//  ================================================================================
//  OPTIONAL EDGE VALIDATIONS (if instrumentation available)
//  ================================================================================
//TEST_SingleTimeoutEvent_EmitsSingleTerminalTransition_NoDoubleFire();
//TEST_LastCommandCompletionTimeStamped_OnTimeoutComplete();
//TEST_ElapsedTimeReported_MatchesApproxTimeoutDuration();

METHOD PRIVATE TEST_Busy_FalseToTrue_OnStart_TrueToFalse_OnComplete
VAR_INST
	DynamicCycles : INT := 0;
END_VAR
VAR
	// Non FB or Interface instance variables
	TestName : Tc2_System.T_MaxString := 'TEST_Busy_FalseToTrue_OnStart_TrueToFalse_OnComplete';
	TestIdx : DINT := INDEX_TEST_BUSY_FALSETOTRUE_ONSTART_TRUETOFALSE_ONCOMPLETE;
	BusyWasTrue : BOOL := FALSE; // Track if we saw Busy=TRUE
END_VAR
TEST(__POUNAME());

// Purpose: Validates Busy flag transitions FALSE→TRUE on start, TRUE→FALSE on complete
// Based on logs: Busy changes at command start (cycle 1,618,132) and timeout complete (cycle 1,618,633)

// Initialize test objects on first cycle only
IF DynamicCycles = 0 THEN
	TestCommand[TestIdx].Initialize();
	TestComponent[TestIdx].Initialize();
	TestCommandConfig[TestIdx].Initialize();
	TestPermIntlk[TestIdx].Initialize();

	// Safe interface assignments
	iTestCommand := TestCommand[TestIdx];
	iTestCommandConfig := TestCommandConfig[TestIdx];
	iTestComponent := TestComponent[TestIdx];
	iTestPermIntlkConfig := TestPermIntlk[TestIdx];

	// Interface validation with protection
	IF iTestCommand = 0 THEN
		AssertTrue(Condition := FALSE, Message := 'TEST FAILED: iTestCommand interface is null');
		DynamicCycles := 0;
		RETURN;
	END_IF

	IF iTestCommandConfig = 0 THEN
		AssertTrue(Condition := FALSE, Message := 'TEST FAILED: iTestCommandConfig interface is null');
		DynamicCycles := 0;
		RETURN;
	END_IF

	IF iTestComponent = 0 THEN
		AssertTrue(Condition := FALSE, Message := 'TEST FAILED: iTestComponent interface is null');
		DynamicCycles := 0;
		RETURN;
	END_IF

	// Configure command to trigger timeout (no completion condition)
	iTestCommandConfig.P_CommandConfiguration.CommandDescription := 'Busy Flag Transition Test';
	iTestCommandConfig.P_CommandConfiguration.TimeoutTime := T#100MS; // Short timeout
	IF __ISVALIDREF(iTestCommandConfig.P_CommandConfiguration.BaseConfiguration) THEN
		iTestCommandConfig.P_CommandConfiguration.BaseConfiguration.LogTraceConfiguration.When := E_LogTraceWhen.xRunOnInitOnly;
	END_IF

	// Setup component to be enabled and not busy
	IF iTestComponent <> 0 THEN
		iTestComponent.P_ComponentStatus.BaseStatus.Enabled := TRUE;
		iTestComponent.P_ComponentStatus.BaseStatus.Busy := FALSE;
		iTestComponent.P_ComponentStatus.BaseStatus.Error := FALSE;
	END_IF

	// Configure permissive to be OK
	IF iTestPermIntlkConfig <> 0 THEN
		iTestPermIntlkConfig.P_PermIntlkConfiguration.PermIntlkObj[1].Description := 'Busy Transition Permissive';
		iTestPermIntlkConfig.P_PermIntlkConfiguration.PermIntlkObj[1].Condition := TRUE;
		iTestPermIntlkConfig.P_PermIntlkConfiguration.PermIntlkObj[1].Index := 1;
		TestPermIntlk[TestIdx].CyclicLogic(); // Update permissive evaluation
	END_IF

	// Setup command with configurations
	iTestCommand.InjectConfigurations(
		iComponent := iTestComponent,
		iCommandConfiguration := iTestCommandConfig,
		iPermIntlkConfiguration := iTestPermIntlkConfig
	);

	// Resolve configurations after injection
	iTestCommand.CyclicLogic();

	// Verify initial Busy is FALSE
	AssertFalse(
		Condition := iTestCommand.P_CommandStatus.BaseStatus.Busy,
		Message := 'Busy should be FALSE before Execute'
	);

	// Execute command
	iTestCommand.Execute();

	// Verify Execute() accepted the command
	AssertEquals_UDINT(
		Expected := E_CommandResult.Accepted,
		Actual := iTestCommand.P_CommandStatus.Result,
		Message := 'Execute() should set Result to Accepted'
	);
ELSE
	// Refresh interface references for subsequent cycles
	iTestCommand := TestCommand[TestIdx];
	iTestCommandConfig := TestCommandConfig[TestIdx];
END_IF

DynamicCycles := DynamicCycles + 1;

// Run cyclic logic
iTestCommand.CyclicLogic();

// Check Busy flag transitions
IF DynamicCycles = 1 THEN
	// After first cycle, Busy should be TRUE (FALSE→TRUE transition)
	AssertTrue(
		Condition := iTestCommand.P_CommandStatus.BaseStatus.Busy,
		Message := 'Busy should transition FALSE→TRUE on command start (cycle 1)'
	);
	BusyWasTrue := TRUE;
END_IF

// Track when Busy goes back to FALSE
IF BusyWasTrue AND NOT iTestCommand.P_CommandStatus.BaseStatus.Busy THEN
	// Busy transitioned TRUE→FALSE (timeout complete)
	AssertEquals_UDINT(
		Expected := E_CommandState.Complete,
		Actual := iTestCommand.P_CommandStatus.StepState,
		Message := 'When Busy transitions TRUE→FALSE, command should be in Complete state'
	);

	// Test passed, finish
	TEST_FINISHED();
END_IF

// Safety: Don't run forever if something goes wrong
IF DynamicCycles > 1000 THEN
	AssertTrue(Condition := FALSE, Message := 'TEST TIMEOUT: Command did not complete after 1000 cycles');
	TEST_FINISHED();
END_IF
END_METHOD

END_FUNCTION_BLOCK

// Tests/FB_LogTests
FUNCTION_BLOCK FB_LogTests EXTENDS TcUnit.FB_TestSuite
VAR
	// Array of test event log handlers - one for each test method
	TestEventLogHandlers : ARRAY[GC_Test.Index_TestFB_Logging_MIN..GC_Test.Index_TestFB_Logging_MAX] OF FB_EventLogHandler;

	// Test instance indices (for clarity and maintainability)
	IDX_FirstCycle					: DINT := 0;
	IDX_NormalOperation				: DINT := 1;
	IDX_BufferHasEntries			: DINT := 2;
	IDX_HighLoad					: DINT := 3;
	IDX_BufferNearCapacity			: DINT := 4;
	IDX_EmergencyFill				: DINT := 5;
	IDX_SuccessfulPersistence		: DINT := 6;
	IDX_FailureOnPersistence		: DINT := 7;
	IDX_RepeatedPersistenceFailures	: DINT := 8;
	IDX_MaxBackoffReached			: DINT := 9;
	IDX_NormalLoadBufferHealth		: DINT := 10;
	IDX_BufferOverflow				: DINT := 11;
	IDX_LogProcessing				: DINT := 12;
	IDX_MultipleCycles				: DINT := 13;
	IDX_ProcessingSeverity			: DINT := 14;
	IDX_TaskCycleExceed			: DINT := 15;
	IDX_TaskWithinLimits			: DINT := 16;
	IDX_AllTasksMonitored			: DINT := 17;
	IDX_EmptyBuffer					: DINT := 18;
	IDX_QueueOverflow				: DINT := 19;

	// Critical test indices
	IDX_PersistenceException		: DINT := 20;
	IDX_PersistenceBlocked			: DINT := 21;
	IDX_BufferNearFullCritical		: DINT := 22;
	IDX_BufferFullCritical			: DINT := 23;
	IDX_MaxDequeueLoad				: DINT := 24;
	IDX_HighJitter					: DINT := 25;
	IDX_ExtendedPersistenceFailure	: DINT := 26;
	IDX_Restart						: DINT := 27;
	IDX_ProcessingAllSeverities	: DINT := 28;
	IDX_OverflowCondition			: DINT := 29;

	// Robustness test indices
	IDX_BufferAtMaxCapacity		: DINT := 30;
	IDX_SustainedHighThroughput	: DINT := 31;
	IDX_MixedSeverityFlood			: DINT := 32;
	IDX_MaxDequeueRate				: DINT := 33;
	IDX_BackoffTimerActive			: DINT := 34;
	IDX_HeavyOSLoad					: DINT := 35;
	IDX_RepeatedPersistenceFailureRobust	: DINT := 36;
	IDX_PersistenceUnhandledException	: DINT := 37;
	IDX_BufferOverflowRecovered		: DINT := 38;
	IDX_MultipleTasksMonitored		: DINT := 39;

	// Note: We have exactly 40 slots (0-39) based on GC_Test configuration
END_VAR

// Core Functional Tests
GivenFirstCycle_WhenProgramRuns_ExpectInitializationComplete();
GivenNormalOperation_WhenLogDequeueCalled_ExpectEntriesProcessed();
GivenBufferHasEntries_WhenDequeueRuns_ExpectEntriesForwarded();
GivenHighLoad_WhenDequeueRuns_ExpectRateReduced();
GivenBufferNearCapacity_WhenDequeueRuns_ExpectRateIncreased();
GivenEmergencyFill_WhenDequeueRuns_ExpectMaxRateCappedAt200();
GivenSuccessfulPersistence_WhenAddToEventLog_ExpectTrueReturned();
GivenFailureOnPersistence_WhenAddToEventLog_ExpectFalseReturned();
GivenRepeatedPersistenceFailures_WhenHandleFailureCalled_ExpectExponentialBackoffApplied();
GivenMaxBackoffReached_WhenHandleFailureCalled_ExpectNoFurtherIncrease();
GivenNormalLoad_WhenUpdateBufferHealthMetrics_ExpectAccurateUtilization();
GivenBufferOverflow_WhenUpdateBufferHealthMetrics_ExpectOverflowCountIncremented();
GivenLogProcessing_WhenUpdatePerformanceMetrics_ExpectThroughputCalculated();
GivenMultipleCycles_WhenUpdatePerformanceMetrics_ExpectRollingAverageUpdated();
GivenProcessing_WhenUpdateSeverityMetrics_ExpectSeverityCountersCorrect();
GivenTaskCycleExceed_WhenMonitorPlcSystemRuns_ExpectCriticalEventLogged();
GivenTaskWithinLimits_WhenMonitorPlcSystemRuns_ExpectNoViolationLogged();
GivenAllTasksMonitored_WhenMonitorPlcSystemRuns_ExpectUtilizationPercentagesCalculated();
GivenEmptyBuffer_WhenLogDequeueCalled_ExpectNoErrors();
GivenQueueOverflow_WhenEnqueueCalled_ExpectOldestEntriesDroppedGracefully();

// High-Criticality Tests
GivenPersistenceThrowsException_WhenAddToEventLog_ExpectSafeRecovery();
GivenPersistenceBlocked_WhenHandleFailureRuns_ExpectProcessingSuspendedUntilTimeout();
GivenBufferNearFull_WhenCriticalAndDebugEntriesEnqueued_ExpectCriticalEntriesPreserved();
GivenBufferFull_WhenNewCriticalEntryArrives_ExpectSpaceReservedForCritical();
GivenMaxDequeueLoad_WhenCycleRuns_ExpectTaskNotToExceed50ms();
GivenHighJitter_WhenMonitoringTaskUtilization_ExpectCorrectHealthScoreLogged();
GivenExtendedPersistenceFailure_WhenRecovered_ExpectRateGraduallyRestored();
GivenRestart_WhenLoggerResumes_ExpectMetricsResetAndSafeStartup();
GivenProcessingAcrossAllSeverities_WhenMetricsUpdated_ExpectAccurateSeverityDistribution();
GivenOverflowCondition_WhenMetricsUpdated_ExpectDroppedCountAccurate();

// Stress and Robustness Tests
GivenBufferAtMaxCapacity_WhenFloodedWithEntries_ExpectGracefulDegradation();
GivenSustainedHighThroughput_WhenRunningFor10Minutes_ExpectNoMemoryLeakOrCycleExceed();
GivenMixedSeverityFlood_WhenProcessing_ExpectLatencyForCriticalEntriesLow();
GivenMaxDequeueRate_WhenCycleRuns_ExpectCycleTimeWithin50msBudget();
GivenBackoffTimerActive_WhenNextCycleRuns_ExpectNoPrematureRetries();
GivenHeavyOSLoad_WhenPersistenceSlows_ExpectLoggerTaskStillMeetsCycleTime();
GivenRepeatedPersistenceFailure_WhenRecovered_ExpectRateRestoredToNormal();
GivenPersistenceThrowsUnhandledException_WhenCaught_ExpectNoTaskCrash();
GivenBufferOverflow_WhenRecovered_ExpectMetricsReflectCorrectDropCounts();
GivenMultipleTasksMonitored_WhenSystemStable_ExpectUtilizationReportedAccurately();
GivenCycleExceeds_WhenDetected_ExpectHealthScoreReducedAndViolationLogged();
GivenSeverityMix_WhenProcessing_ExpectSeverityDistributionAccurate();

METHOD PRIVATE GivenAllTasksMonitored_WhenMonitorPlcSystemRuns_ExpectUtilizationPercentagesCalculated
VAR
END_VAR
TEST(__POUNAME());

//Assertions

TEST_FINISHED();
END_METHOD

METHOD PRIVATE GivenBufferHasEntries_WhenDequeueRuns_ExpectEntriesForwarded
VAR
	TestHandler				: REFERENCE TO FB_EventLogHandler;
	InitialBufferCount		: UDINT;
	FinalBufferCount		: UDINT;
	i						: INT;
	EntriesAdded			: INT := 10;
	ExpectedProcessed		: UDINT;
	ActualProcessed			: UDINT;
END_VAR
TEST(__POUNAME());

// Get reference to test instance for this test
TestHandler REF= TestEventLogHandlers[IDX_BufferHasEntries];

// Configure test instance for test mode
IF __ISVALIDREF(TestHandler.P_EventLogHandlerConfiguration.BaseConfiguration) THEN
	TestHandler.P_EventLogHandlerConfiguration.BaseConfiguration.InSimulation := TRUE;
ELSE
	TestHandler.Initialize();
END_IF

// Initialize the test handler and system components
TestHandler.Initialize();
GVL_System.RingBufferLog.Initialize();
GVL_System.GlobalEventLog.Initialize();

// Call CyclicLogic to process initialization
TestHandler.CyclicLogic();

// Ensure clean state
GVL_System.RingBufferLog.ClearBuffer();

// Arrange - Add entries to the buffer
InitialBufferCount := GVL_System.RingBufferLog.P_RingBufferStatus.ObjectCountInBufferPrim;

// Add test entries to buffer
FOR i := 1 TO EntriesAdded DO
	GVL_System.RingBufferLog.TraceWithSeverity(
		Message := CONCAT('Entry to forward #', INT_TO_STRING(i)),
		Severity := Global.TcEventSeverity.Info
	);
END_FOR

// Verify entries were added to buffer
AssertEquals_UDINT(
	Expected := InitialBufferCount + INT_TO_UDINT(EntriesAdded),
	Actual := GVL_System.RingBufferLog.P_RingBufferStatus.ObjectCountInBufferPrim,
	Message := 'Entries should be added to buffer before dequeue'
);

// Store the initial processed count
ActualProcessed := TestHandler.P_EventLogHandlerStatus.LoggingMetrics.TotalEntriesProcessed;

// Act - Run CyclicLogic which will dequeue and forward entries
TestHandler.CyclicLogic();

// Get final state
FinalBufferCount := GVL_System.RingBufferLog.P_RingBufferStatus.ObjectCountInBufferPrim;
ActualProcessed := TestHandler.P_EventLogHandlerStatus.LogCountThisScan;

// Assert - Verify entries were removed from buffer
AssertTrue(
	Condition := FinalBufferCount < InitialBufferCount + INT_TO_UDINT(EntriesAdded),
	Message := 'Buffer count should decrease after dequeue'
);

// Verify entries were actually processed (forwarded)
AssertTrue(
	Condition := ActualProcessed > 0,
	Message := 'Entries should be processed (forwarded) during dequeue'
);

// Calculate expected processed based on dynamic rate limits
ExpectedProcessed := MIN(INT_TO_UDINT(EntriesAdded),
                         UINT_TO_UDINT(TestHandler.P_EventLogHandlerStatus.DynamicMaxEntries));

// Verify we didn't exceed the dynamic rate limit
AssertTrue(
	Condition := ActualProcessed <= UINT_TO_UDINT(TestHandler.P_EventLogHandlerStatus.DynamicMaxEntries),
	Message := 'Should not process more than DynamicMaxEntries in one scan'
);

// Verify the number of entries removed matches the number processed
AssertEquals_UDINT(
	Expected := ActualProcessed,
	Actual := (InitialBufferCount + INT_TO_UDINT(EntriesAdded)) - FinalBufferCount,
	Message := 'Number of entries removed from buffer should match number processed'
);

// Verify metrics were updated
AssertEquals_UDINT(
	Expected := ActualProcessed,
	Actual := UINT_TO_UDINT(TestHandler.P_EventLogHandlerStatus.LoggingMetrics.EntriesProcessedThisCycle),
	Message := 'EntriesProcessedThisCycle should match actual processed count'
);

// Verify total entries processed was incremented
AssertTrue(
	Condition := TestHandler.P_EventLogHandlerStatus.LoggingMetrics.TotalEntriesProcessed >= ActualProcessed,
	Message := 'TotalEntriesProcessed should be incremented'
);

// Verify no errors during forwarding
AssertFalse(
	Condition := TestHandler.P_EventLogHandlerStatus.BaseStatus.Error,
	Message := 'No errors should occur during normal forwarding operation'
);

// Verify buffer health metrics were updated
AssertTrue(
	Condition := TestHandler.P_EventLogHandlerStatus.LoggingMetrics.BufferUtilizationPercentage >= 0.0,
	Message := 'Buffer utilization should be calculated after dequeue'
);

TEST_FINISHED();
END_METHOD

METHOD PRIVATE GivenBufferNearCapacity_WhenDequeueRuns_ExpectRateIncreased
VAR
	TestHandler				: REFERENCE TO FB_EventLogHandler;
	BufferCapacity			: UDINT;
	EntriesToAdd			: UDINT;
	NormalRate				: UINT;
	IncreasedRate			: UINT;
	i						: DINT;
	InitialBufferCount		: UDINT;
	FinalBufferCount		: UDINT;
	EntriesProcessed		: UDINT;
END_VAR
TEST(__POUNAME());

// Get reference to test instance for this test
TestHandler REF= TestEventLogHandlers[IDX_BufferNearCapacity];

// Configure test instance - enable metrics tracking

// Initialize the test handler and system components
TestHandler.Initialize();
GVL_System.RingBufferLog.Initialize();
GVL_System.GlobalEventLog.Initialize();

// Call CyclicLogic to process initialization
TestHandler.CyclicLogic();

// Ensure clean state
GVL_System.RingBufferLog.ClearBuffer();

// Get buffer capacity
BufferCapacity := GVL_System.RingBufferLog.P_RingBufferStatus.BufferCapacity;

// Arrange - Set low task utilization (so rate increase is based on buffer, not task load)
GVL_System.PlcSystemInfo[GPL_BASE.INDEX_LOG_TASK].TaskUtilizationPercentage := 0.2; // 20% utilization

// Calculate normal rate with empty buffer
NormalRate := TestHandler.CalculateDynamicRate();

// Verify we're at normal rate with low load and empty buffer
AssertEquals_UINT(
	Expected := UDINT_TO_UINT(GPL_Base.MAX_LOG_ENTRIES_PER_SCAN),
	Actual := NormalRate,
	Message := 'Low load with empty buffer should use normal rate'
);

// Fill buffer to near capacity (80% full - should trigger rate increase)
EntriesToAdd := (BufferCapacity * 80) / 100;  // 80% of capacity

FOR i := 1 TO UDINT_TO_DINT(EntriesToAdd) DO
	GVL_System.RingBufferLog.TraceWithSeverity(
		Message := CONCAT('Buffer fill test entry ', DINT_TO_STRING(i)),
		Severity := Global.TcEventSeverity.Info
	);
END_FOR

InitialBufferCount := GVL_System.RingBufferLog.P_RingBufferStatus.ObjectCountInBufferPrim;

// Verify buffer is near capacity
AssertTrue(
	Condition := InitialBufferCount >= (BufferCapacity * 75) / 100,
	Message := 'Buffer should be at least 75% full for this test'
);

// Act - Calculate rate with near-full buffer
IncreasedRate := TestHandler.CalculateDynamicRate();

// Assert - Rate should be increased when buffer is near capacity
AssertTrue(
	Condition := IncreasedRate > NormalRate,
	Message := 'Processing rate should increase when buffer is near capacity'
);

// Specifically, when buffer > 75% and low task load, rate should double
AssertEquals_UINT(
	Expected := UDINT_TO_UINT(GPL_Base.MAX_LOG_ENTRIES_PER_SCAN * 2),
	Actual := IncreasedRate,
	Message := 'Buffer near capacity with low load should double the rate'
);

// Verify the increased rate doesn't exceed emergency maximum
AssertTrue(
	Condition := IncreasedRate <= UDINT_TO_UINT(200),
	Message := 'Increased rate should not exceed emergency maximum'
);

// Call CyclicLogic to process with increased rate
TestHandler.CyclicLogic();

// Get final state
FinalBufferCount := GVL_System.RingBufferLog.P_RingBufferStatus.ObjectCountInBufferPrim;
EntriesProcessed := TestHandler.P_EventLogHandlerStatus.LogCountThisScan;

// Verify more entries were processed with increased rate
AssertTrue(
	Condition := EntriesProcessed > UINT_TO_UDINT(NormalRate),
	Message := 'Should process more entries when rate is increased'
);

// Verify buffer was reduced
AssertTrue(
	Condition := FinalBufferCount < InitialBufferCount,
	Message := 'Buffer count should decrease after processing with increased rate'
);

// Test emergency fill level (>90%)
GVL_System.RingBufferLog.ClearBuffer();
EntriesToAdd := (BufferCapacity * 95) / 100;  // 95% of capacity

FOR i := 1 TO UDINT_TO_DINT(EntriesToAdd) DO
	GVL_System.RingBufferLog.TraceWithSeverity(
		Message := CONCAT('Emergency fill test ', DINT_TO_STRING(i)),
		Severity := Global.TcEventSeverity.Critical
	);
END_FOR

// Calculate rate with emergency fill level
IncreasedRate := TestHandler.CalculateDynamicRate();

// Should be at emergency maximum
AssertEquals_UINT(
	Expected := UDINT_TO_UINT(200),
	Actual := IncreasedRate,
	Message := 'Emergency fill level should trigger maximum processing rate'
);

TEST_FINISHED();
END_METHOD

METHOD PRIVATE GivenBufferOverflow_WhenUpdateBufferHealthMetrics_ExpectOverflowCountIncremented
VAR
	InitialOverflowCount		: UDINT;
	FinalOverflowCount			: UDINT;
	BufferCapacity				: UDINT;
	i							: DINT;
	TestBufferFull				: BOOL;
END_VAR
TEST(__POUNAME());

// Initialize if needed
IF GVL_System.PlcSystemInfo[GPL_Base.INDEX_LOG_TASK].FirstCycle THEN
    GVL_System.RingBufferLog.Initialize();
    GVL_System.GlobalEventLog.Initialize();
    RETURN;
END_IF;

// Arrange - Get initial state
InitialOverflowCount := GVL_System.EventLogHandler.P_EventLogHandlerStatus.LoggingMetrics.BufferOverflowCount;
BufferCapacity := GVL_System.RingBufferLog.P_RingBufferStatus.BufferCapacity;

// Clear the buffer first
GVL_System.RingBufferLog.ClearBuffer();

// Fill the buffer to capacity
FOR i := 1 TO UDINT_TO_DINT(BufferCapacity) + 10 DO
	GVL_System.RingBufferLog.TraceWithSeverity(
		Message := CONCAT('Overflow test entry ', DINT_TO_STRING(i)),
		Severity := Global.TcEventSeverity.Info
	);
END_FOR;

// Verify buffer is full
TestBufferFull := GVL_System.RingBufferLog.P_RingBufferStatus.BufferIsFullPrim;
AssertTrue(
	Condition := TestBufferFull,
	Message := 'Buffer should be full after adding more entries than capacity'
);

// Act - Call UpdateBufferHealthMetrics multiple times while buffer is full
GVL_System.EventLogHandler.UpdateBufferHealthMetrics();  // First call - should increment
GVL_System.EventLogHandler.UpdateBufferHealthMetrics();  // Second call - should NOT increment (edge detection)
GVL_System.EventLogHandler.UpdateBufferHealthMetrics();  // Third call - should NOT increment

FinalOverflowCount := GVL_System.EventLogHandler.P_EventLogHandlerStatus.LoggingMetrics.BufferOverflowCount;

// Assert - Overflow count should increment only once due to edge detection
AssertEquals_UDINT(
	Expected := InitialOverflowCount + 1,
	Actual := FinalOverflowCount,
	Message := 'Overflow count should increment only once on rising edge of buffer full'
);

// Clear some entries to make buffer not full
// Call LogDequeue multiple times to ensure buffer is drained enough
FOR i := 1 TO 10 DO
	GVL_System.EventLogHandler.LogDequeue();
	IF NOT GVL_System.RingBufferLog.P_RingBufferStatus.BufferIsFullPrim THEN
		EXIT; // Buffer is no longer full, stop dequeuing
	END_IF;
END_FOR;

// Reset the edge trigger by having buffer not full
TestBufferFull := GVL_System.RingBufferLog.P_RingBufferStatus.BufferIsFullPrim;
AssertFalse(
	Condition := TestBufferFull,
	Message := 'Buffer should not be full after dequeue'
);

// Fill again to test another edge
FOR i := 1 TO 100 DO
	GVL_System.RingBufferLog.TraceWithSeverity(
		Message := CONCAT('Second overflow test ', DINT_TO_STRING(i)),
		Severity := Global.TcEventSeverity.Critical
	);
END_FOR;

// Call UpdateBufferHealthMetrics again with new overflow
GVL_System.EventLogHandler.UpdateBufferHealthMetrics();

// Should increment again on new rising edge
AssertEquals_UDINT(
	Expected := InitialOverflowCount + 2,
	Actual := GVL_System.EventLogHandler.P_EventLogHandlerStatus.LoggingMetrics.BufferOverflowCount,
	Message := 'Overflow count should increment on each new rising edge'
);

TEST_FINISHED();
END_METHOD

METHOD PRIVATE GivenEmergencyFill_WhenDequeueRuns_ExpectMaxRateCappedAt200
VAR
END_VAR
TEST(__POUNAME());

//Assertions

TEST_FINISHED();
END_METHOD

METHOD PRIVATE GivenEmptyBuffer_WhenLogDequeueCalled_ExpectNoErrors
VAR
	TestHandler					: REFERENCE TO FB_EventLogHandler;
	InitialErrorState			: BOOL;
	FinalErrorState				: BOOL;
	InitialProcessedCount		: UDINT;
	FinalProcessedCount			: UDINT;
	BufferCountBeforeDequeue	: UDINT;
	BufferCountAfterDequeue	: UDINT;
END_VAR
TEST(__POUNAME());

// Get reference to test instance for this test
TestHandler REF= TestEventLogHandlers[IDX_EmptyBuffer];

// Configure test instance - enable metrics tracking

// Initialize the test handler and system components
TestHandler.Initialize();
GVL_System.RingBufferLog.Initialize();
GVL_System.GlobalEventLog.Initialize();

// Call CyclicLogic to process initialization
TestHandler.CyclicLogic();

// Ensure buffer is completely empty
GVL_System.RingBufferLog.ClearBuffer();

// Verify buffer is empty
AssertEquals_UDINT(
	Expected := 0,
	Actual := GVL_System.RingBufferLog.P_RingBufferStatus.ObjectCountInBufferPrim,
	Message := 'Buffer should be empty before test'
);

// Get initial state
InitialErrorState := TestHandler.P_EventLogHandlerStatus.BaseStatus.Error;
InitialProcessedCount := TestHandler.P_EventLogHandlerStatus.LoggingMetrics.TotalEntriesProcessed;
BufferCountBeforeDequeue := GVL_System.RingBufferLog.P_RingBufferStatus.ObjectCountInBufferPrim;

// Verify no errors initially
AssertFalse(
	Condition := InitialErrorState,
	Message := 'Should start with no errors'
);

// Act - Call LogDequeue on empty buffer (should handle gracefully)
TestHandler.LogDequeue();

// Get final state
FinalErrorState := TestHandler.P_EventLogHandlerStatus.BaseStatus.Error;
FinalProcessedCount := TestHandler.P_EventLogHandlerStatus.LoggingMetrics.TotalEntriesProcessed;
BufferCountAfterDequeue := GVL_System.RingBufferLog.P_RingBufferStatus.ObjectCountInBufferPrim;

// Assert - No errors should occur
AssertFalse(
	Condition := FinalErrorState,
	Message := 'No errors should occur when dequeuing from empty buffer'
);

// Buffer should remain empty
AssertEquals_UDINT(
	Expected := 0,
	Actual := BufferCountAfterDequeue,
	Message := 'Buffer should remain empty'
);

// No entries should be processed
AssertEquals_UDINT(
	Expected := InitialProcessedCount,
	Actual := FinalProcessedCount,
	Message := 'No entries should be processed from empty buffer'
);

// LogCountThisScan should be 0
AssertEquals_UDINT(
	Expected := 0,
	Actual := TestHandler.P_EventLogHandlerStatus.LogCountThisScan,
	Message := 'LogCountThisScan should be 0 for empty buffer'
);

// Test multiple dequeue calls on empty buffer (should all handle gracefully)
TestHandler.LogDequeue();
TestHandler.LogDequeue();
TestHandler.LogDequeue();

// Still no errors
AssertFalse(
	Condition := TestHandler.P_EventLogHandlerStatus.BaseStatus.Error,
	Message := 'Multiple dequeue calls on empty buffer should not cause errors'
);

// Call full CyclicLogic on empty buffer (should handle gracefully)
TestHandler.CyclicLogic();

// Verify no errors after full cycle
AssertFalse(
	Condition := TestHandler.P_EventLogHandlerStatus.BaseStatus.Error,
	Message := 'Full CyclicLogic on empty buffer should not cause errors'
);

// Verify metrics remain stable
AssertEquals_UDINT(
	Expected := 0,
	Actual := TestHandler.P_EventLogHandlerStatus.LoggingMetrics.EntriesProcessedThisCycle,
	Message := 'EntriesProcessedThisCycle should be 0 for empty buffer'
);

// Buffer utilization should be 0%
AssertEquals_REAL(
	Expected := 0.0,
	Actual := TestHandler.P_EventLogHandlerStatus.LoggingMetrics.BufferUtilizationPercentage,
	Delta := 0.01,
	Message := 'Buffer utilization should be 0% when empty'
);

// Dynamic rate calculation should still work
AssertTrue(
	Condition := TestHandler.CalculateDynamicRate() > 0,
	Message := 'Dynamic rate calculation should work even with empty buffer'
);

// No persistence failures should occur
AssertEquals_UINT(
	Expected := 0,
	Actual := TestHandler.P_EventLogHandlerStatus.BackoffState.PersistenceFailureCount,
	Message := 'No persistence failures should occur with empty buffer'
);

// System health should be good
AssertTrue(
	Condition := TestHandler.P_EventLogHandlerStatus.LoggingMetrics.SystemHealthScore >= 90.0,
	Message := 'System health should be high with empty buffer and no errors'
);

TEST_FINISHED();
END_METHOD

METHOD PRIVATE GivenFailureOnPersistence_WhenAddToEventLog_ExpectFalseReturned
VAR
	TestHandler				: REFERENCE TO FB_EventLogHandler;
	PersistenceResult		: BOOL;
	InitialSuccessCount		: UDINT;
	FinalSuccessCount		: UDINT;
	InitialFailureCount		: UINT;
	FinalFailureCount		: UINT;
END_VAR
TEST(__POUNAME());

// Get reference to test instance for this test
TestHandler REF= TestEventLogHandlers[IDX_FailureOnPersistence];

// Configure test instance for TEST MODE to simulate failure
IF __ISVALIDREF(TestHandler.P_EventLogHandlerConfiguration.BaseConfiguration) THEN
	TestHandler.P_EventLogHandlerConfiguration.BaseConfiguration.InSimulation := TRUE;
ELSE
	TestHandler.Initialize();
END_IF

// Initialize the test handler and system components
TestHandler.Initialize();
GVL_System.RingBufferLog.Initialize();
GVL_System.GlobalEventLog.Initialize();

// Call CyclicLogic to process initialization
TestHandler.CyclicLogic();

// Ensure clean state
GVL_System.RingBufferLog.ClearBuffer();

// Get initial metrics
InitialFailureCount := TestHandler.P_EventLogHandlerStatus.BackoffState.PersistenceFailureCount;

// Arrange - Simulate a persistence failure condition
// Since we're in test mode, we need to mock the failure
// This would require setting up the test status to simulate failure
TestHandler.P_EventLogHandlerStatus.BackoffState.PersistenceBlocked := TRUE;

// Add a test entry to the buffer
GVL_System.RingBufferLog.TraceWithSeverity(
	Message := 'Test entry for failed persistence',
	Severity := Global.TcEventSeverity.Error
);

// Verify entry was added
AssertEquals_UDINT(
	Expected := 1,
	Actual := GVL_System.RingBufferLog.P_RingBufferStatus.ObjectCountInBufferPrim,
	Message := 'One entry should be in buffer'
);

// Act - Try to add to event log when persistence is blocked
// First, remove from buffer to make available in P_LastObjectRemoved
GVL_System.RingBufferLog.RemoveObject();

// Now try to add it to the event log (should fail due to PersistenceBlocked)
PersistenceResult := TestHandler.AddToEventLog();

// Assert - Verify failed persistence
AssertFalse(
	Condition := PersistenceResult,
	Message := 'AddToEventLog should return FALSE when persistence is blocked'
);

// Get final metrics
FinalFailureCount := TestHandler.P_EventLogHandlerStatus.BackoffState.PersistenceFailureCount;

// Success count verification removed as PersistenceSuccessCount metric doesn't exist

// Reset persistence blocked to test normal failure handling
TestHandler.P_EventLogHandlerStatus.BackoffState.PersistenceBlocked := FALSE;

// Simulate a different type of failure - we could mock the GlobalEventLog to fail
// For this test, we'll simulate by checking the behavior when AddToEventLog
// is called but the operation fails (returns FALSE)

// Add another entry
GVL_System.RingBufferLog.TraceWithSeverity(
	Message := 'Test entry for simulated add failure',
	Severity := Global.TcEventSeverity.Critical
);

// Process it
GVL_System.RingBufferLog.RemoveObject();

// In test mode, we can force AddToEventLog to return FALSE
// by manipulating the test status - this simulates GlobalEventLog failure
// Note: This assumes AddToEventLog checks some condition we can control
// If not, we'd need a method to simulate GlobalEventLog failures

// Call HandlePersistenceFailure to simulate what happens on failure
TestHandler.HandlePersistenceFailure();

// Verify failure handling was activated
AssertTrue(
	Condition := TestHandler.P_EventLogHandlerStatus.BackoffState.PersistenceBlocked,
	Message := 'Persistence should be blocked after handling failure'
);

// Verify backoff delay was set
AssertTrue(
	Condition := TestHandler.P_EventLogHandlerStatus.BackoffState.BackoffDelayMs >= 100,
	Message := 'Backoff delay should be set after failure'
);

// Verify failure count incremented
AssertTrue(
	Condition := TestHandler.P_EventLogHandlerStatus.BackoffState.PersistenceFailureCount > 0,
	Message := 'PersistenceFailureCount should increment after failure'
);

// Backoff timer check removed as BackoffStartTime property doesn't exist

TEST_FINISHED();
END_METHOD

METHOD PRIVATE GivenFirstCycle_WhenProgramRuns_ExpectInitializationComplete
VAR
	// Local test variables
	PreInitBufferCount		: UDINT;
	PostInitBufferCount		: UDINT;
	TestHandler				: REFERENCE TO FB_EventLogHandler;
END_VAR
TEST(__POUNAME());

// Get reference to test instance for this test
TestHandler REF= TestEventLogHandlers[IDX_FirstCycle];

// Configure test instance for test mode
IF __ISVALIDREF(TestHandler.P_EventLogHandlerConfiguration.BaseConfiguration) THEN
	TestHandler.P_EventLogHandlerConfiguration.BaseConfiguration.InSimulation := TRUE;
ELSE
	TestHandler.Initialize();
END_IF

// Configure test instance settings

// Initialize the test instance
TestHandler.Initialize();

// Call CyclicLogic to process initialization
TestHandler.CyclicLogic();

// Arrange - Clear any existing state and store pre-init values
GVL_System.RingBufferLog.ClearBuffer();
PreInitBufferCount := GVL_System.RingBufferLog.P_RingBufferStatus.ObjectCountInBufferPrim;

// Act - Simulate what the EventLogHandler does on first cycle:
// Initialize both the RingBufferLog and GlobalEventLog
GVL_System.RingBufferLog.Initialize();
GVL_System.GlobalEventLog.Initialize();
PostInitBufferCount := GVL_System.RingBufferLog.P_RingBufferStatus.ObjectCountInBufferPrim;

// Verify the test handler is initialized
AssertTrue(
	Condition := TestHandler.P_EventLogHandlerStatus.BaseStatus.Initialized,
	Message := 'Test EventLogHandler should be initialized'
);

// Assert - Verify components are properly initialized
AssertTrue(
	Condition := __ISVALIDREF(GVL_System.RingBufferLog.P_RingBufferStatus.BaseStatus) AND
	             GVL_System.RingBufferLog.P_RingBufferStatus.BaseStatus.Initialized,
	Message := 'RingBufferLog should be initialized after first cycle behavior'
);

AssertTrue(
	Condition := GVL_System.GlobalEventLog.P_BaseStatus.Initialized,
	Message := 'GlobalEventLog should be initialized after first cycle behavior'
);

// Verify ring buffer is ready for dequeue operations
AssertEquals_UDINT(
	Expected := 0,
	Actual := PostInitBufferCount,
	Message := 'RingBufferLog should be empty and ready for entries after initialization'
);

// Verify buffer has proper capacity configured
AssertTrue(
	Condition := GVL_System.RingBufferLog.P_RingBufferStatus.BufferCapacity > 0,
	Message := 'RingBufferLog must have a positive capacity to accept log entries'
);

// Verify no error states that would prevent dequeue operations
AssertFalse(
	Condition := __ISVALIDREF(GVL_System.RingBufferLog.P_RingBufferStatus.BaseStatus) AND
	             GVL_System.RingBufferLog.P_RingBufferStatus.BaseStatus.Error,
	Message := 'No errors should be present that would block dequeue operations'
);

AssertFalse(
	Condition := GVL_System.RingBufferLog.P_RingBufferStatus.BufferIsFullPrim,
	Message := 'Buffer should not report full state after initialization'
);

// Verify global event log has no errors that would prevent receiving entries
AssertFalse(
	Condition := GVL_System.GlobalEventLog.P_BaseStatus.Error,
	Message := 'GlobalEventLog should have no errors that would prevent receiving dequeued entries'
);

// Verify test handler configuration is in test mode
IF __ISVALIDREF(TestHandler.P_EventLogHandlerConfiguration.BaseConfiguration) THEN
	AssertTrue(
		Condition := TestHandler.P_EventLogHandlerConfiguration.BaseConfiguration.InSimulation,
		Message := 'EventLogHandler should be in test mode'
	);
ELSE
	AssertTrue(
		Condition := FALSE,
		Message := 'EventLogHandlerConfiguration reference is invalid - cannot verify test mode'
	);
END_IF

// Verify test handler metrics are initialized
AssertEquals_UDINT(
	Expected := 0,
	Actual := TestHandler.P_EventLogHandlerStatus.LoggingMetrics.TotalEntriesProcessed,
	Message := 'Total entries processed should be 0 after initialization'
);

AssertEquals_REAL(
	Expected := 100.0,
	Actual := TestHandler.P_EventLogHandlerStatus.LoggingMetrics.SystemHealthScore,
	Delta := 0.01,
	Message := 'System health score should be 100% after initialization'
);

TEST_FINISHED();
END_METHOD

METHOD PRIVATE GivenHighLoad_WhenDequeueRuns_ExpectRateReduced
VAR
	TestHandler					: REFERENCE TO FB_EventLogHandler;
	SimulatedHighUtilization	: REAL := 0.85;  // 85% utilization
	SimulatedNormalUtilization	: REAL := 0.30;  // 30% utilization
	NormalMaxEntries			: UINT;
	HighLoadMaxEntries			: UINT;
	i							: INT;
	InitialBufferCount			: UDINT;
	FinalBufferCount			: UDINT;
	EntriesProcessed			: UDINT;
END_VAR
TEST(__POUNAME());

// Get reference to test instance for this test
TestHandler REF= TestEventLogHandlers[IDX_HighLoad];

// Configure test instance for test mode
IF __ISVALIDREF(TestHandler.P_EventLogHandlerConfiguration.BaseConfiguration) THEN
	TestHandler.P_EventLogHandlerConfiguration.BaseConfiguration.InSimulation := TRUE;
ELSE
	TestHandler.Initialize();
END_IF

// Initialize the test handler and system components
TestHandler.Initialize();
GVL_System.RingBufferLog.Initialize();
GVL_System.GlobalEventLog.Initialize();

// Call CyclicLogic to process initialization
TestHandler.CyclicLogic();

// Ensure clean state
GVL_System.RingBufferLog.ClearBuffer();

// Arrange - Set up normal load condition first
GVL_System.PlcSystemInfo[GPL_BASE.INDEX_LOG_TASK].TaskUtilizationPercentage := SimulatedNormalUtilization;

// Calculate normal rate by calling CalculateDynamicRate
NormalMaxEntries := TestHandler.CalculateDynamicRate();

// Verify normal rate is at expected level
AssertEquals_UINT(
	Expected := UDINT_TO_UINT(GPL_Base.MAX_LOG_ENTRIES_PER_SCAN),
	Actual := NormalMaxEntries,
	Message := 'Normal load should allow full processing rate'
);

// Now simulate high load condition
GVL_System.PlcSystemInfo[GPL_BASE.INDEX_LOG_TASK].TaskUtilizationPercentage := SimulatedHighUtilization;

// Add many entries to process
FOR i := 1 TO 50 DO
	GVL_System.RingBufferLog.TraceWithSeverity(
		Message := CONCAT('High load test entry ', INT_TO_STRING(i)),
		Severity := Global.TcEventSeverity.Warning
	);
END_FOR

InitialBufferCount := GVL_System.RingBufferLog.P_RingBufferStatus.ObjectCountInBufferPrim;

// Act - Calculate dynamic rate under high load
HighLoadMaxEntries := TestHandler.CalculateDynamicRate();

// Assert - Rate should be reduced under high load
AssertTrue(
	Condition := HighLoadMaxEntries < NormalMaxEntries,
	Message := 'Processing rate should be reduced under high load'
);

// When utilization > LOG_CYCLE_EXCEED_MAX_THRESHOLD (0.75), rate should be quartered
AssertEquals_UINT(
	Expected := UDINT_TO_UINT(GPL_Base.MAX_LOG_ENTRIES_PER_SCAN / 4),
	Actual := HighLoadMaxEntries,
	Message := 'High load (>75%) should reduce rate to quarter of normal'
);

// Store the calculated rate in the test handler's status
TestHandler.P_EventLogHandlerStatus.DynamicMaxEntries := HighLoadMaxEntries;

// Call CyclicLogic to process with the high load condition
TestHandler.CyclicLogic();

// Get final state
FinalBufferCount := GVL_System.RingBufferLog.P_RingBufferStatus.ObjectCountInBufferPrim;
EntriesProcessed := TestHandler.P_EventLogHandlerStatus.LogCountThisScan;

// Verify it respects the reduced rate limit
AssertTrue(
	Condition := EntriesProcessed <= UINT_TO_UDINT(HighLoadMaxEntries),
	Message := 'Should not process more than reduced rate limit under high load'
);

// Verify that entries were actually processed (but at reduced rate)
AssertTrue(
	Condition := EntriesProcessed > 0 AND EntriesProcessed <= UINT_TO_UDINT(HighLoadMaxEntries),
	Message := 'Should process some entries but respect high load limit'
);

// Verify buffer count decreased by the amount processed
AssertEquals_UDINT(
	Expected := InitialBufferCount - EntriesProcessed,
	Actual := FinalBufferCount,
	Message := 'Buffer should decrease by exactly the number of entries processed'
);

// Test moderate load (between 50% and 75%)
GVL_System.PlcSystemInfo[GPL_BASE.INDEX_LOG_TASK].TaskUtilizationPercentage := 0.6; // 60% utilization
NormalMaxEntries := TestHandler.CalculateDynamicRate();

// Should be half rate for moderate load
AssertEquals_UINT(
	Expected := UDINT_TO_UINT(GPL_Base.MAX_LOG_ENTRIES_PER_SCAN / 2),
	Actual := NormalMaxEntries,
	Message := 'Moderate load (50-75%) should reduce rate to half of normal'
);

TEST_FINISHED();
END_METHOD

METHOD PRIVATE GivenLogProcessing_WhenUpdatePerformanceMetrics_ExpectThroughputCalculated
VAR
END_VAR
TEST(__POUNAME());

//Assertions

TEST_FINISHED();
END_METHOD

METHOD PRIVATE GivenMaxBackoffReached_WhenHandleFailureCalled_ExpectNoFurtherIncrease
VAR
END_VAR
TEST(__POUNAME());

//Assertions

TEST_FINISHED();
END_METHOD

METHOD PRIVATE GivenMultipleCycles_WhenUpdatePerformanceMetrics_ExpectRollingAverageUpdated
VAR
	TestHandler					: REFERENCE TO FB_EventLogHandler;
	InitialAverage				: REAL;
	PreviousAverage				: REAL;
	CurrentAverage				: REAL;
	i							: INT;
	j							: INT;
	NumCycles					: INT := 10;
	EntriesPerCycle				: INT := 5;
	AverageChanged				: BOOL := FALSE;
	PeakTime					: UDINT;
END_VAR
TEST(__POUNAME());

// Get reference to test instance for this test
TestHandler REF= TestEventLogHandlers[IDX_MultipleCycles];

// Configure test instance - enable performance metrics

// Initialize the test handler and system components
TestHandler.Initialize();
GVL_System.RingBufferLog.Initialize();
GVL_System.GlobalEventLog.Initialize();

// Call CyclicLogic to process initialization
TestHandler.CyclicLogic();

// Ensure clean state
GVL_System.RingBufferLog.ClearBuffer();

// Get initial average (should be 0 or very low after init)
InitialAverage := TestHandler.P_EventLogHandlerStatus.LoggingMetrics.AverageProcessingTimeMs;

// Store initial value
PreviousAverage := InitialAverage;

// Act - Run multiple cycles with entries to process
FOR i := 1 TO NumCycles DO

	// Add entries for this cycle
	FOR j := 1 TO EntriesPerCycle DO
		GVL_System.RingBufferLog.TraceWithSeverity(
			Message := CONCAT('Cycle ', CONCAT(INT_TO_STRING(i), CONCAT(' Entry ', INT_TO_STRING(j)))),
			Severity := Global.TcEventSeverity.Info
		);
	END_FOR

	// Process the entries
	TestHandler.CyclicLogic();

	// Get current average after this cycle
	CurrentAverage := TestHandler.P_EventLogHandlerStatus.LoggingMetrics.AverageProcessingTimeMs;

	// Check if average has changed (it should update with each cycle)
	IF CurrentAverage <> PreviousAverage THEN
		AverageChanged := TRUE;
	END_IF

	// Store for next iteration
	PreviousAverage := CurrentAverage;

END_FOR

// Assert - Rolling average should have been updated
AssertTrue(
	Condition := AverageChanged,
	Message := 'Rolling average should update across multiple cycles'
);

// Average should be a reasonable positive value after processing
AssertTrue(
	Condition := CurrentAverage > 0.0,
	Message := 'Average processing time should be positive after multiple cycles'
);

// Average should not be exactly the initial value (unless it was 0 and stayed 0, which would be wrong)
AssertTrue(
	Condition := CurrentAverage <> InitialAverage OR InitialAverage = 0.0,
	Message := 'Average should change from initial value after processing'
);

// Test that average is actually an average (not just the last value)
// Add a cycle with many more entries (should affect average)
FOR j := 1 TO 50 DO
	GVL_System.RingBufferLog.TraceWithSeverity(
		Message := CONCAT('Heavy cycle entry ', INT_TO_STRING(j)),
		Severity := Global.TcEventSeverity.Warning
	);
END_FOR

PreviousAverage := CurrentAverage;
TestHandler.CyclicLogic();
CurrentAverage := TestHandler.P_EventLogHandlerStatus.LoggingMetrics.AverageProcessingTimeMs;

// Average should have changed with the heavier cycle
AssertTrue(
	Condition := CurrentAverage <> PreviousAverage,
	Message := 'Average should adjust when processing time changes significantly'
);

// Verify rolling average weights are being applied
// The new average should be between the old average and the new measurement
// (This assumes RollingAvgWeightPrevious + RollingAvgWeightCurrent = 1.0)
IF __ISVALIDREF(TestHandler.P_EventLogHandlerConfiguration) THEN
	AssertTrue(
		Condition := TestHandler.P_EventLogHandlerConfiguration.RollingAvgWeightPrevious +
		             TestHandler.P_EventLogHandlerConfiguration.RollingAvgWeightCurrent <= 1.01 AND
		             TestHandler.P_EventLogHandlerConfiguration.RollingAvgWeightPrevious +
		             TestHandler.P_EventLogHandlerConfiguration.RollingAvgWeightCurrent >= 0.99,
		Message := 'Rolling average weights should sum to approximately 1.0'
	);
ELSE
	AssertTrue(
		Condition := FALSE,
		Message := 'EventLogHandlerConfiguration reference is invalid - cannot verify rolling average weights'
	);
END_IF

// Peak time should also be tracked
PeakTime := TestHandler.P_EventLogHandlerStatus.LoggingMetrics.PeakProcessingTimeMs;
AssertTrue(
	Condition := PeakTime > 0,
	Message := 'Peak processing time should be tracked'
);

// Peak should be >= average (peak is the maximum, average is... average)
AssertTrue(
	Condition := UDINT_TO_REAL(PeakTime) >= CurrentAverage,
	Message := 'Peak time should be greater than or equal to average time'
);

// Test with empty buffer cycles (should still update average)
GVL_System.RingBufferLog.ClearBuffer();
PreviousAverage := CurrentAverage;

FOR i := 1 TO 3 DO
	TestHandler.CyclicLogic();  // Process with empty buffer
END_FOR

CurrentAverage := TestHandler.P_EventLogHandlerStatus.LoggingMetrics.AverageProcessingTimeMs;

// Average should trend towards lower values with empty buffer processing
// (empty cycles should be faster)
AssertTrue(
	Condition := CurrentAverage <= PreviousAverage + 0.1,  // Allow small tolerance
	Message := 'Average should decrease or stay similar when processing empty buffer'
);

// Verify other performance metrics are also updated
AssertTrue(
	Condition := TestHandler.P_EventLogHandlerStatus.LoggingMetrics.TotalEntriesProcessed > 0,
	Message := 'Total entries processed should be tracked'
);

AssertTrue(
	Condition := TestHandler.P_EventLogHandlerStatus.LoggingMetrics.CycleUtilizationPercentage >= 0.0,
	Message := 'Cycle utilization should be calculated'
);

TEST_FINISHED();
END_METHOD

METHOD PRIVATE GivenNormalLoad_WhenUpdateBufferHealthMetrics_ExpectAccurateUtilization
VAR
END_VAR
TEST(__POUNAME());

//Assertions

TEST_FINISHED();
END_METHOD

METHOD PRIVATE GivenNormalOperation_WhenLogDequeueCalled_ExpectEntriesProcessed
VAR
	TestHandler		: REFERENCE TO FB_EventLogHandler;
	InitialCount	: UDINT;
	FinalCount		: UDINT;
	i				: INT;
	TestMessage		: STRING := 'Test log entry';
	InitialTotalProcessed	: UDINT;
	FinalTotalProcessed		: UDINT;
END_VAR
TEST(__POUNAME());

// Get reference to test instance for this test
TestHandler REF= TestEventLogHandlers[IDX_NormalOperation];

// Configure test instance for test mode
IF __ISVALIDREF(TestHandler.P_EventLogHandlerConfiguration.BaseConfiguration) THEN
	TestHandler.P_EventLogHandlerConfiguration.BaseConfiguration.InSimulation := TRUE;
ELSE
	TestHandler.Initialize();
END_IF

// Initialize the test handler and system components
TestHandler.Initialize();
GVL_System.RingBufferLog.Initialize();
GVL_System.GlobalEventLog.Initialize();

// Ensure clean state
GVL_System.RingBufferLog.ClearBuffer();

// Arrange - Store initial state
InitialCount := GVL_System.RingBufferLog.P_RingBufferStatus.ObjectCountInBufferPrim;
InitialTotalProcessed := TestHandler.P_EventLogHandlerStatus.LoggingMetrics.TotalEntriesProcessed;

// Add 5 test entries with different severities
GVL_System.RingBufferLog.TraceWithSeverity(
	Message := CONCAT(TestMessage, ' 1 - Info'),
	Severity := Global.TcEventSeverity.Info
);
GVL_System.RingBufferLog.TraceWithSeverity(
	Message := CONCAT(TestMessage, ' 2 - Warning'),
	Severity := Global.TcEventSeverity.Warning
);
GVL_System.RingBufferLog.TraceWithSeverity(
	Message := CONCAT(TestMessage, ' 3 - Error'),
	Severity := Global.TcEventSeverity.Error
);
GVL_System.RingBufferLog.TraceWithSeverity(
	Message := CONCAT(TestMessage, ' 4 - Critical'),
	Severity := Global.TcEventSeverity.Critical
);
GVL_System.RingBufferLog.TraceWithSeverity(
	Message := CONCAT(TestMessage, ' 5 - Info'),
	Severity := Global.TcEventSeverity.Info
);

// Verify entries were added
AssertEquals_UDINT(
	Expected := InitialCount + 5,
	Actual := GVL_System.RingBufferLog.P_RingBufferStatus.ObjectCountInBufferPrim,
	Message := '5 entries should be added to buffer'
);

// Capture buffer count before calling CyclicLogic (MonitorPlcSystem may add entries)
InitialCount := GVL_System.RingBufferLog.P_RingBufferStatus.ObjectCountInBufferPrim;

// Act - Call CyclicLogic which will internally call LogDequeue and update metrics
TestHandler.CyclicLogic();

// Assert - Check that entries were processed
FinalCount := GVL_System.RingBufferLog.P_RingBufferStatus.ObjectCountInBufferPrim;
FinalTotalProcessed := TestHandler.P_EventLogHandlerStatus.LoggingMetrics.TotalEntriesProcessed;

AssertTrue(
	Condition := FinalCount < InitialCount,
	Message := 'Buffer count should decrease after dequeue'
);

// Verify the handler processed entries
AssertTrue(
	Condition := TestHandler.P_EventLogHandlerStatus.LogCountThisScan > 0,
	Message := 'LogCountThisScan should be greater than 0 after processing'
);

// Verify metrics consistency
AssertEquals_UDINT(
	Expected := TestHandler.P_EventLogHandlerStatus.LogCountThisScan,
	Actual := UINT_TO_UDINT(TestHandler.P_EventLogHandlerStatus.LoggingMetrics.EntriesProcessedThisCycle),
	Message := 'EntriesProcessedThisCycle should match LogCountThisScan'
);

// Verify total entries processed was incremented
AssertTrue(
	Condition := FinalTotalProcessed > InitialTotalProcessed,
	Message := 'TotalEntriesProcessed should increase after processing'
);

// Verify the actual number of entries processed
AssertEquals_UDINT(
	Expected := InitialCount - FinalCount,
	Actual := TestHandler.P_EventLogHandlerStatus.LogCountThisScan,
	Message := 'LogCountThisScan should equal the number of entries removed from buffer'
);

// Verify buffer utilization metrics were updated
AssertTrue(
	Condition := TestHandler.P_EventLogHandlerStatus.LoggingMetrics.BufferUtilizationPercentage >= 0.0,
	Message := 'Buffer utilization should be calculated'
);

// Verify severity tracking if enabled
	// At least some severity counters should have been incremented
	AssertTrue(
		Condition := (TestHandler.P_EventLogHandlerStatus.LoggingMetrics.InfoEntriesProcessed +
					  TestHandler.P_EventLogHandlerStatus.LoggingMetrics.WarningEntriesProcessed +
					  TestHandler.P_EventLogHandlerStatus.LoggingMetrics.ErrorEntriesProcessed +
					  TestHandler.P_EventLogHandlerStatus.LoggingMetrics.CriticalEntriesProcessed) > 0,
		Message := 'Severity counters should be incremented when processing entries'
	);

// Verify no errors occurred during processing
AssertFalse(
	Condition := TestHandler.P_EventLogHandlerStatus.BaseStatus.Error,
	Message := 'No errors should occur during normal dequeue operation'
);

// Verify dynamic rate was calculated
AssertTrue(
	Condition := TestHandler.P_EventLogHandlerStatus.DynamicMaxEntries > 0,
	Message := 'Dynamic max entries should be calculated and positive'
);

TEST_FINISHED();
END_METHOD

METHOD PRIVATE GivenProcessing_WhenUpdateSeverityMetrics_ExpectSeverityCountersCorrect
VAR
END_VAR
TEST(__POUNAME());

//Assertions

TEST_FINISHED();
END_METHOD

METHOD PRIVATE GivenQueueOverflow_WhenEnqueueCalled_ExpectOldestEntriesDroppedGracefully
VAR
	TestHandler				: REFERENCE TO FB_EventLogHandler;
	BufferCapacity			: UDINT;
	i						: DINT;
	FirstEntryMessage		: STRING := 'FIRST_ENTRY_MARKER';
	LastEntryMessage		: STRING := 'LAST_ENTRY_MARKER';
	OverflowMessage			: STRING := 'OVERFLOW_ENTRY';
	InitialBufferCount		: UDINT;
	FinalBufferCount		: UDINT;
	InitialOverflowCount	: UDINT;
	FinalOverflowCount		: UDINT;
	ProcessedEntry			: BOOL;
END_VAR
TEST(__POUNAME());

// Get reference to test instance for this test
TestHandler REF= TestEventLogHandlers[IDX_QueueOverflow];

// Configure test instance - enable metrics tracking

// Initialize the test handler and system components
TestHandler.Initialize();
GVL_System.RingBufferLog.Initialize();
GVL_System.GlobalEventLog.Initialize();

// Call CyclicLogic to process initialization
TestHandler.CyclicLogic();

// Ensure clean state
GVL_System.RingBufferLog.ClearBuffer();

// Get buffer capacity
BufferCapacity := GVL_System.RingBufferLog.P_RingBufferStatus.BufferCapacity;

// Get initial metrics
InitialOverflowCount := TestHandler.P_EventLogHandlerStatus.LoggingMetrics.BufferOverflowCount;

// Arrange - Fill buffer to capacity with numbered entries
// Add a recognizable first entry
GVL_System.RingBufferLog.TraceWithSeverity(
	Message := FirstEntryMessage,
	Severity := Global.TcEventSeverity.Info
);

// Fill the rest of the buffer
FOR i := 2 TO UDINT_TO_DINT(BufferCapacity - 1) DO
	GVL_System.RingBufferLog.TraceWithSeverity(
		Message := CONCAT('Queue entry #', DINT_TO_STRING(i)),
		Severity := Global.TcEventSeverity.Info
	);
END_FOR

// Add a recognizable last entry before overflow
GVL_System.RingBufferLog.TraceWithSeverity(
	Message := LastEntryMessage,
	Severity := Global.TcEventSeverity.Warning
);

// Verify buffer is at capacity
AssertEquals_UDINT(
	Expected := BufferCapacity,
	Actual := GVL_System.RingBufferLog.P_RingBufferStatus.ObjectCountInBufferPrim,
	Message := 'Buffer should be at full capacity'
);

InitialBufferCount := GVL_System.RingBufferLog.P_RingBufferStatus.ObjectCountInBufferPrim;

// Act - Try to enqueue when buffer is full (should handle gracefully)
// This should either drop the oldest entry or reject the new one
GVL_System.RingBufferLog.TraceWithSeverity(
	Message := OverflowMessage,
	Severity := Global.TcEventSeverity.Critical
);

// Update metrics to detect overflow
TestHandler.UpdateBufferHealthMetrics();

// Get final state
FinalBufferCount := GVL_System.RingBufferLog.P_RingBufferStatus.ObjectCountInBufferPrim;
FinalOverflowCount := TestHandler.P_EventLogHandlerStatus.LoggingMetrics.BufferOverflowCount;

// Assert - Buffer handled overflow gracefully
AssertTrue(
	Condition := FinalBufferCount <= BufferCapacity,
	Message := 'Buffer count should not exceed capacity'
);

// Overflow should have been detected
AssertEquals_UDINT(
	Expected := InitialOverflowCount + 1,
	Actual := FinalOverflowCount,
	Message := 'Overflow count should increment'
);

// No errors should occur
AssertFalse(
	Condition := TestHandler.P_EventLogHandlerStatus.BaseStatus.Error,
	Message := 'No errors should occur during overflow handling'
);

// Process some entries to check what remains
TestHandler.CyclicLogic();

// If ring buffer drops oldest, the first entry should be gone
// If it rejects new entries, the overflow entry should not be present
// Either way, system should remain stable

// Test multiple overflow attempts
FOR i := 1 TO 10 DO
	GVL_System.RingBufferLog.TraceWithSeverity(
		Message := CONCAT('Additional overflow ', DINT_TO_STRING(i)),
		Severity := Global.TcEventSeverity.Info
	);
END_FOR

// Update metrics multiple times
TestHandler.UpdateBufferHealthMetrics();
TestHandler.UpdateBufferHealthMetrics();

// Should still be stable
AssertFalse(
	Condition := TestHandler.P_EventLogHandlerStatus.BaseStatus.Error,
	Message := 'Multiple overflow attempts should not cause errors'
);

// Buffer should still be within limits
AssertTrue(
	Condition := GVL_System.RingBufferLog.P_RingBufferStatus.ObjectCountInBufferPrim <= BufferCapacity,
	Message := 'Buffer should never exceed capacity even after multiple overflow attempts'
);

// Test recovery - clear some space and verify normal operation resumes
TestHandler.CyclicLogic();  // Process some entries
TestHandler.CyclicLogic();  // Process more

// Should have some space now
AssertTrue(
	Condition := GVL_System.RingBufferLog.P_RingBufferStatus.ObjectCountInBufferPrim < BufferCapacity,
	Message := 'Buffer should have space after processing'
);

// Add new entries - should work normally
GVL_System.RingBufferLog.TraceWithSeverity(
	Message := 'Post-overflow normal entry',
	Severity := Global.TcEventSeverity.Info
);

// Verify it was added
AssertTrue(
	Condition := GVL_System.RingBufferLog.P_RingBufferStatus.ObjectCountInBufferPrim > 0,
	Message := 'Should be able to add entries after overflow recovery'
);

// System health should remain reasonable despite overflow
AssertTrue(
	Condition := TestHandler.P_EventLogHandlerStatus.LoggingMetrics.SystemHealthScore > 0.0,
	Message := 'System health should remain positive even after overflow'
);

// Verify buffer utilization metrics are accurate
AssertTrue(
	Condition := TestHandler.P_EventLogHandlerStatus.LoggingMetrics.BufferUtilizationPercentage >= 0.0 AND
	             TestHandler.P_EventLogHandlerStatus.LoggingMetrics.BufferUtilizationPercentage <= 100.0,
	Message := 'Buffer utilization should be within 0-100% range'
);

TEST_FINISHED();
END_METHOD

METHOD PRIVATE GivenRepeatedPersistenceFailures_WhenHandleFailureCalled_ExpectExponentialBackoffApplied
VAR
	ExpectedDelays	: ARRAY[1..7] OF UDINT := [100, 200, 400, 800, 1600, 3200, 10000];
	i				: INT;
	InitialBackoffCount	: UDINT;
END_VAR
TEST(__POUNAME());

// Initialize if needed
IF GVL_System.PlcSystemInfo[GPL_Base.INDEX_LOG_TASK].FirstCycle THEN
    GVL_System.RingBufferLog.Initialize();
    GVL_System.GlobalEventLog.Initialize();
    RETURN;
END_IF;

// Arrange - Cannot directly reset backoff state due to encapsulation
// Test may need to be restructured to work with the new architecture
// For now, we'll work with whatever the current state is
InitialBackoffCount := GVL_System.EventLogHandler.P_EventLogHandlerStatus.LoggingMetrics.BackoffActiveCount;

// Act & Assert - Simulate successive failures and verify exponential backoff
FOR i := 1 TO 7 DO
	// Simulate a persistence failure
	GVL_System.EventLogHandler.HandlePersistenceFailure();

	// Assert correct backoff delay for this failure count
	AssertEquals_UDINT(
		Expected := ExpectedDelays[i],
		Actual := GVL_System.EventLogHandler.P_EventLogHandlerStatus.BackoffState.BackoffDelayMs,
		Message := CONCAT('Backoff delay should be ', UDINT_TO_STRING(ExpectedDelays[i]))
	);

	// Verify persistence is blocked
	AssertTrue(
		Condition := GVL_System.EventLogHandler.P_EventLogHandlerStatus.BackoffState.PersistenceBlocked,
		Message := 'Persistence should be blocked after failure'
	);

	// Verify failure count
	AssertEquals_UINT(
		Expected := INT_TO_UINT(i),
		Actual := GVL_System.EventLogHandler.P_EventLogHandlerStatus.BackoffState.PersistenceFailureCount,
		Message := CONCAT('Failure count should be ', INT_TO_STRING(i))
	);
END_FOR;

// Verify backoff activations were counted (one per failure)
AssertEquals_UDINT(
	Expected := InitialBackoffCount + 7,
	Actual := GVL_System.EventLogHandler.P_EventLogHandlerStatus.LoggingMetrics.BackoffActiveCount,
	Message := 'BackoffActiveCount should increment for each activation'
);

// Test that further failures stay at max backoff
GVL_System.EventLogHandler.HandlePersistenceFailure(); // 8th failure
AssertEquals_UDINT(
	Expected := 10000,  // Should stay at max
	Actual := GVL_System.EventLogHandler.P_EventLogHandlerStatus.BackoffState.BackoffDelayMs,
	Message := 'Backoff should be capped at 10000ms'
);

// NOTE: Cannot directly reset PersistenceFailureCount due to encapsulation
// The test for reset behavior after success cannot be performed without
// a way to reset the internal state or a method that simulates success
// PRG_LOG.EventLogHandler.BackoffState.PersistenceFailureCount := 0;  // NOT ALLOWED
// PRG_LOG.EventLogHandler.HandlePersistenceFailure();
// AssertEquals_UDINT(Expected := 100, Actual := ..., Message := 'Reset test cannot be performed');

TEST_FINISHED();
END_METHOD

METHOD PRIVATE GivenSuccessfulPersistence_WhenAddToEventLog_ExpectTrueReturned
VAR
	TestHandler				: REFERENCE TO FB_EventLogHandler;
	PersistenceResult		: BOOL;
	InitialSuccessCount		: UDINT;
	FinalSuccessCount		: UDINT;
	InitialFailureCount		: UINT;
	FinalFailureCount		: UINT;
END_VAR
TEST(__POUNAME());

// Get reference to test instance for this test
TestHandler REF= TestEventLogHandlers[IDX_SuccessfulPersistence];

// Configure test instance - enable metrics tracking

// Initialize the test handler and system components
TestHandler.Initialize();
GVL_System.RingBufferLog.Initialize();
GVL_System.GlobalEventLog.Initialize();

// Call CyclicLogic to process initialization
TestHandler.CyclicLogic();

// Ensure clean state
GVL_System.RingBufferLog.ClearBuffer();

// Get initial metrics
InitialFailureCount := TestHandler.P_EventLogHandlerStatus.BackoffState.PersistenceFailureCount;

// Arrange - Add a test entry to the buffer using TestHandler.TraceWithSeverity
// (TraceWithSeverity adds to GVL_System.RingBufferLog)
TestHandler.TraceWithSeverity(
	Message := 'Test entry for successful persistence',
	Severity := Global.TcEventSeverity.Info
);

// Verify entry was added
AssertEquals_UDINT(
	Expected := 1,
	Actual := GVL_System.RingBufferLog.P_RingBufferStatus.ObjectCountInBufferPrim,
	Message := 'One entry should be in buffer'
);

// Act - Dequeue the entry which will attempt to persist it
// First, we need to remove it from the buffer so it's available in P_LastObjectRemoved
GVL_System.RingBufferLog.RemoveObject();

// Now try to add it to the event log
PersistenceResult := TestHandler.AddToEventLog();

// Assert - Verify successful persistence
AssertTrue(
	Condition := PersistenceResult,
	Message := 'AddToEventLog should return TRUE for successful persistence'
);

// Get final metrics
FinalFailureCount := TestHandler.P_EventLogHandlerStatus.BackoffState.PersistenceFailureCount;

// Without PersistenceSuccessCount metric, we rely on the return value to verify success

// Verify failure count was not incremented
AssertEquals_UINT(
	Expected := InitialFailureCount,
	Actual := FinalFailureCount,
	Message := 'PersistenceFailureCount should not change on successful persistence'
);

// Verify no backoff is active
AssertFalse(
	Condition := TestHandler.P_EventLogHandlerStatus.BackoffState.PersistenceBlocked,
	Message := 'Persistence should not be blocked after successful operation'
);

// Verify backoff delay is at minimum (or zero)
AssertTrue(
	Condition := TestHandler.P_EventLogHandlerStatus.BackoffState.BackoffDelayMs <= 100,
	Message := 'Backoff delay should be minimal after successful persistence'
);

// Test multiple successful persistences
// Add and process several more entries
FOR InitialSuccessCount := 1 TO 3 DO
	GVL_System.RingBufferLog.TraceWithSeverity(
		Message := CONCAT('Additional test entry ', UDINT_TO_STRING(InitialSuccessCount)),
		Severity := Global.TcEventSeverity.Warning
	);
END_FOR

// Process all entries via CyclicLogic
TestHandler.CyclicLogic();

// Multiple successes verified through CyclicLogic processing

// Verify total entries processed increased
AssertTrue(
	Condition := TestHandler.P_EventLogHandlerStatus.LoggingMetrics.TotalEntriesProcessed > 0,
	Message := 'TotalEntriesProcessed should increase with successful persistence'
);

TEST_FINISHED();
END_METHOD

METHOD PRIVATE GivenTaskCycleExceed_WhenMonitorPlcSystemRuns_ExpectCriticalEventLogged
VAR
	InitialBufferCount		: UDINT;
	FinalBufferCount		: UDINT;
	TestTaskIndex			: DINT := 2;  // Use a test task index
	InitialHealthScore		: REAL;
	FinalHealthScore		: REAL;
END_VAR
TEST(__POUNAME());

// Initialize if needed
IF GVL_System.PlcSystemInfo[GPL_Base.INDEX_LOG_TASK].FirstCycle THEN
    GVL_System.RingBufferLog.Initialize();
    GVL_System.GlobalEventLog.Initialize();
    RETURN;
END_IF;

// Arrange - Set up initial state
GVL_System.RingBufferLog.ClearBuffer();
InitialBufferCount := GVL_System.RingBufferLog.P_RingBufferStatus.ObjectCountInBufferPrim;

// Ensure task index is within bounds
IF TestTaskIndex > UPPER_BOUND(GVL_System.PlcSystemInfo, 1) THEN
	TestTaskIndex := 1;
END_IF;

// Reset the edge trigger first by ensuring CycleTimeExceeded is FALSE
GVL_System.PlcSystemInfo[TestTaskIndex].CycleTimeExceeded := FALSE;
GVL_System.EventLogHandler.MonitorPlcSystem();  // Call once with FALSE to reset trigger

// Get initial health score
InitialHealthScore := GVL_System.EventLogHandler.P_EventLogHandlerStatus.LoggingMetrics.SystemHealthScore;

// Act - Simulate a cycle exceed condition
GVL_System.PlcSystemInfo[TestTaskIndex].CycleTimeExceeded := TRUE;

// Call MonitorPlcSystem which should detect the edge and log
GVL_System.EventLogHandler.MonitorPlcSystem();

// Get final buffer count
FinalBufferCount := GVL_System.RingBufferLog.P_RingBufferStatus.ObjectCountInBufferPrim;

// Assert - A critical log entry should have been added
AssertEquals_UDINT(
	Expected := InitialBufferCount + 1,
	Actual := FinalBufferCount,
	Message := 'One critical entry should be logged for cycle exceed'
);

// Verify the logged entry is critical severity
IF FinalBufferCount > InitialBufferCount THEN
	// The last entry should be the cycle exceed message
	// Note: We can't directly check the severity without dequeuing,
	// but we can verify the log was created
	AssertTrue(
		Condition := TRUE,
		Message := 'Cycle exceed event was logged'
	);
END_IF;

// Call MonitorPlcSystem again with same state - should NOT log again (edge detection)
GVL_System.EventLogHandler.MonitorPlcSystem();
AssertEquals_UDINT(
	Expected := FinalBufferCount,  // Should not change
	Actual := GVL_System.RingBufferLog.P_RingBufferStatus.ObjectCountInBufferPrim,
	Message := 'No duplicate log on sustained cycle exceed (edge detection working)'
);

// Note: UpdatePerformanceMetrics is now a protected method (_UpdatePerformanceMetrics)
// and cannot be called directly from tests. The health score update would normally
// happen internally during the CyclicLogic execution.
// PRG_LOG.EventLogHandler.UpdatePerformanceMetrics(ULINT_TO_UDINT(Tc2_System.F_GetSystemTime()));
FinalHealthScore := GVL_System.EventLogHandler.P_EventLogHandlerStatus.LoggingMetrics.SystemHealthScore;

// Health score check disabled since UpdatePerformanceMetrics is now protected
// and we cannot directly test the health score update from cycle exceed.
// AssertTrue(
// 	Condition := FinalHealthScore < InitialHealthScore,
// //	Message := 'Health score should decrease when cycle exceed is detected'
// );

// Reset cycle exceed and verify edge reset works
GVL_System.PlcSystemInfo[TestTaskIndex].CycleTimeExceeded := FALSE;
GVL_System.EventLogHandler.MonitorPlcSystem();

// Set cycle exceed again - should log again after reset
GVL_System.PlcSystemInfo[TestTaskIndex].CycleTimeExceeded := TRUE;
GVL_System.EventLogHandler.MonitorPlcSystem();

AssertEquals_UDINT(
	Expected := FinalBufferCount + 1,
	Actual := GVL_System.RingBufferLog.P_RingBufferStatus.ObjectCountInBufferPrim,
	Message := 'New cycle exceed should be logged after reset'
);

TEST_FINISHED();
END_METHOD

METHOD PRIVATE GivenTaskWithinLimits_WhenMonitorPlcSystemRuns_ExpectNoViolationLogged
VAR
END_VAR
TEST(__POUNAME());

//Assertions

TEST_FINISHED();
END_METHOD

METHOD PRIVATE GivenBufferFull_WhenNewCriticalEntryArrives_ExpectSpaceReservedForCritical
VAR
END_VAR
TEST(__POUNAME());

//Assertions

TEST_FINISHED();
END_METHOD

METHOD PRIVATE GivenBufferNearFull_WhenCriticalAndDebugEntriesEnqueued_ExpectCriticalEntriesPreserved
VAR
END_VAR
TEST(__POUNAME());

//Assertions

TEST_FINISHED();
END_METHOD

METHOD PRIVATE GivenExtendedPersistenceFailure_WhenRecovered_ExpectRateGraduallyRestored
VAR
END_VAR
TEST(__POUNAME());

//Assertions

TEST_FINISHED();
END_METHOD

METHOD PRIVATE GivenHighJitter_WhenMonitoringTaskUtilization_ExpectCorrectHealthScoreLogged
VAR
END_VAR
TEST(__POUNAME());

//Assertions

TEST_FINISHED();
END_METHOD

METHOD PRIVATE GivenMaxDequeueLoad_WhenCycleRuns_ExpectTaskNotToExceed50ms
VAR
	TestHandler				: REFERENCE TO FB_EventLogHandler;
	BufferCapacity			: UDINT;
	i						: DINT;
	StartTime				: ULINT;
	EndTime					: ULINT;
	ProcessingTimeMs		: UDINT;
	MaxAllowedTimeMs		: UDINT := 50;  // 50ms budget
	EntriesProcessed		: UDINT;
	MaxEntriesToAdd			: UDINT;
END_VAR
TEST(__POUNAME());

// Get reference to test instance for this test
TestHandler REF= TestEventLogHandlers[IDX_MaxDequeueLoad];

// Configure test instance - enable performance metrics to track timing

// Initialize the test handler and system components
TestHandler.Initialize();
GVL_System.RingBufferLog.Initialize();
GVL_System.GlobalEventLog.Initialize();

// Call CyclicLogic to process initialization
TestHandler.CyclicLogic();

// Ensure clean state
GVL_System.RingBufferLog.ClearBuffer();

// Get buffer capacity and determine max load
BufferCapacity := GVL_System.RingBufferLog.P_RingBufferStatus.BufferCapacity;

// Fill buffer to maximum capacity to create worst-case load
MaxEntriesToAdd := MIN(BufferCapacity, UINT_TO_UDINT(200));

FOR i := 1 TO UDINT_TO_DINT(MaxEntriesToAdd) DO
	GVL_System.RingBufferLog.TraceWithSeverity(
		Message := CONCAT('Max load test entry ', DINT_TO_STRING(i)),
		Severity := Global.TcEventSeverity.Info
	);
END_FOR

// Verify buffer has entries to process
AssertTrue(
	Condition := GVL_System.RingBufferLog.P_RingBufferStatus.ObjectCountInBufferPrim > 0,
	Message := 'Buffer should have entries for max load test'
);

// Act - Measure processing time for maximum dequeue load
StartTime := Tc2_System.F_GetSystemTime();

// Process maximum allowed entries in one cycle
TestHandler.CyclicLogic();

EndTime := Tc2_System.F_GetSystemTime();

// Calculate processing time in milliseconds
ProcessingTimeMs := ULINT_TO_UDINT((EndTime - StartTime) / 10000);  // Convert from 100ns units to ms

// Get number of entries processed
EntriesProcessed := TestHandler.P_EventLogHandlerStatus.LogCountThisScan;

// Assert - Processing time should not exceed 50ms budget
AssertTrue(
	Condition := ProcessingTimeMs <= MaxAllowedTimeMs,
	Message := CONCAT('Processing time should not exceed 50ms. Actual: ', UDINT_TO_STRING(ProcessingTimeMs))
);

// Verify entries were actually processed
AssertTrue(
	Condition := EntriesProcessed > 0,
	Message := 'Entries should be processed during the cycle'
);

// Verify dynamic rate limiting is working
AssertTrue(
	Condition := EntriesProcessed <= UINT_TO_UDINT(TestHandler.P_EventLogHandlerStatus.DynamicMaxEntries),
	Message := 'Should not exceed dynamic max entries per scan'
);

// Check peak processing time metric
AssertTrue(
	Condition := TestHandler.P_EventLogHandlerStatus.LoggingMetrics.PeakProcessingTimeMs <= MaxAllowedTimeMs,
	Message := 'Peak processing time metric should not exceed 50ms'
);

// Test with emergency fill level to ensure rate limiting prevents timeout
GVL_System.RingBufferLog.ClearBuffer();

// Fill to emergency level (95% of capacity)
MaxEntriesToAdd := (BufferCapacity * 95) / 100;

FOR i := 1 TO UDINT_TO_DINT(MaxEntriesToAdd) DO
	GVL_System.RingBufferLog.TraceWithSeverity(
		Message := CONCAT('Emergency load test ', DINT_TO_STRING(i)),
		Severity := Global.TcEventSeverity.Critical
	);
END_FOR

// Set low task utilization to allow maximum processing rate
GVL_System.PlcSystemInfo[GPL_BASE.INDEX_LOG_TASK].TaskUtilizationPercentage := 0.1;

// Measure emergency processing
StartTime := Tc2_System.F_GetSystemTime();
TestHandler.CyclicLogic();
EndTime := Tc2_System.F_GetSystemTime();

ProcessingTimeMs := ULINT_TO_UDINT((EndTime - StartTime) / 10000);
EntriesProcessed := TestHandler.P_EventLogHandlerStatus.LogCountThisScan;

// Even at emergency rate, should not exceed time budget
AssertTrue(
	Condition := ProcessingTimeMs <= MaxAllowedTimeMs,
	Message := CONCAT('Emergency processing should not exceed 50ms. Actual: ', UDINT_TO_STRING(ProcessingTimeMs))
);

// Verify emergency rate was used
AssertTrue(
	Condition := EntriesProcessed <= UINT_TO_UDINT(200),
	Message := 'Should not exceed emergency max entries'
);

// Test high CPU load scenario - should reduce rate to stay within budget
GVL_System.PlcSystemInfo[GPL_BASE.INDEX_LOG_TASK].TaskUtilizationPercentage := 0.9;  // 90% utilization

// Calculate expected reduced rate
TestHandler.CalculateDynamicRate();

// Process with high load
StartTime := Tc2_System.F_GetSystemTime();
TestHandler.CyclicLogic();
EndTime := Tc2_System.F_GetSystemTime();

ProcessingTimeMs := ULINT_TO_UDINT((EndTime - StartTime) / 10000);

// Should still stay within budget due to rate reduction
AssertTrue(
	Condition := ProcessingTimeMs <= MaxAllowedTimeMs,
	Message := CONCAT('High load processing should stay within 50ms due to rate reduction. Actual: ', UDINT_TO_STRING(ProcessingTimeMs))
);

// Verify average processing time is reasonable
AssertTrue(
	Condition := TestHandler.P_EventLogHandlerStatus.LoggingMetrics.AverageProcessingTimeMs <= UDINT_TO_REAL(MaxAllowedTimeMs),
	Message := 'Average processing time should be within budget'
);

TEST_FINISHED();
END_METHOD

METHOD PRIVATE GivenOverflowCondition_WhenMetricsUpdated_ExpectDroppedCountAccurate
VAR
	TestHandler				: REFERENCE TO FB_EventLogHandler;
	BufferCapacity			: UDINT;
	InitialDroppedCount		: UDINT;
	FinalDroppedCount		: UDINT;
	InitialOverflowCount	: UDINT;
	FinalOverflowCount		: UDINT;
	i						: DINT;
	EntriesToOverfill		: UDINT;
	ExpectedDropped			: UDINT;
END_VAR
TEST(__POUNAME());

// Get reference to test instance for this test
TestHandler REF= TestEventLogHandlers[IDX_OverflowCondition];

// Configure test instance - enable metrics tracking

// Initialize the test handler and system components
TestHandler.Initialize();
GVL_System.RingBufferLog.Initialize();
GVL_System.GlobalEventLog.Initialize();

// Call CyclicLogic to process initialization
TestHandler.CyclicLogic();

// Ensure clean state
GVL_System.RingBufferLog.ClearBuffer();

// Get buffer capacity
BufferCapacity := GVL_System.RingBufferLog.P_RingBufferStatus.BufferCapacity;

// Get initial metrics
InitialOverflowCount := TestHandler.P_EventLogHandlerStatus.LoggingMetrics.BufferOverflowCount;

// Arrange - Fill buffer to capacity first
FOR i := 1 TO UDINT_TO_DINT(BufferCapacity) DO
	GVL_System.RingBufferLog.TraceWithSeverity(
		Message := CONCAT('Fill buffer entry ', DINT_TO_STRING(i)),
		Severity := Global.TcEventSeverity.Info
	);
END_FOR

// Verify buffer is full
AssertTrue(
	Condition := GVL_System.RingBufferLog.P_RingBufferStatus.BufferIsFullPrim,
	Message := 'Buffer should be full before testing overflow'
);

// Now try to add more entries (these should be dropped)
EntriesToOverfill := 10;
FOR i := 1 TO UDINT_TO_DINT(EntriesToOverfill) DO
	GVL_System.RingBufferLog.TraceWithSeverity(
		Message := CONCAT('Overflow entry ', DINT_TO_STRING(i)),
		Severity := Global.TcEventSeverity.Warning
	);
END_FOR

// Act - Update buffer health metrics to detect overflow
TestHandler.UpdateBufferHealthMetrics();

// Get final metrics
FinalOverflowCount := TestHandler.P_EventLogHandlerStatus.LoggingMetrics.BufferOverflowCount;

// Assert - Verify overflow was detected
AssertEquals_UDINT(
	Expected := InitialOverflowCount + 1,
	Actual := FinalOverflowCount,
	Message := 'BufferOverflowCount should increment when overflow detected'
);

// The actual dropped count depends on the ring buffer implementation
// If it's a circular buffer, old entries might be overwritten
// If it rejects new entries when full, the new ones are dropped
// We need to check what actually happened

IF GVL_System.RingBufferLog.P_RingBufferStatus.ObjectCountInBufferPrim = BufferCapacity THEN
	// Buffer stayed at capacity - new entries were rejected/dropped
	ExpectedDropped := EntriesToOverfill;

	// Note: The dropped count might need to be tracked differently
	// depending on how the RingBuffer handles overflow
	AssertTrue(
		Condition := FinalDroppedCount >= InitialDroppedCount,
		Message := 'Dropped count should increase or stay same when entries are rejected'
	);
ELSE
	// Buffer might have wrapped around or handled overflow differently
	AssertTrue(
		Condition := TRUE,
		Message := 'Overflow condition was handled'
	);
END_IF

// Test severity-specific drop tracking
GVL_System.RingBufferLog.ClearBuffer();

// Fill with mixed severity entries
FOR i := 1 TO UDINT_TO_DINT(BufferCapacity - 5) DO
	GVL_System.RingBufferLog.TraceWithSeverity(
		Message := CONCAT('Info entry ', DINT_TO_STRING(i)),
		Severity := Global.TcEventSeverity.Info
	);
END_FOR

// Add some critical entries (these should be preserved if possible)
FOR i := 1 TO 5 DO
	GVL_System.RingBufferLog.TraceWithSeverity(
		Message := CONCAT('Critical entry ', DINT_TO_STRING(i)),
		Severity := Global.TcEventSeverity.Critical
	);
END_FOR

// Buffer should be full now
AssertTrue(
	Condition := GVL_System.RingBufferLog.P_RingBufferStatus.BufferIsFullPrim,
	Message := 'Buffer should be full with mixed severities'
);

// Try to add more non-critical entries (should be dropped in favor of critical)
FOR i := 1 TO 5 DO
	GVL_System.RingBufferLog.TraceWithSeverity(
		Message := CONCAT('Additional info entry ', DINT_TO_STRING(i)),
		Severity := Global.TcEventSeverity.Info
	);
END_FOR

// Update metrics again
TestHandler.UpdateBufferHealthMetrics();

// Verify metrics reflect the overflow condition
AssertTrue(
	Condition := TestHandler.P_EventLogHandlerStatus.LoggingMetrics.BufferUtilizationPercentage >= 95.0,
	Message := 'Buffer utilization should be very high during overflow'
);

// Process some entries to clear space
TestHandler.CyclicLogic();

// After processing, dropped count metrics should be maintained
AssertTrue(
	Condition := TestHandler.P_EventLogHandlerStatus.LoggingMetrics.BufferOverflowCount > 0,
	Message := 'Overflow count should persist after processing'
);

// Verify the system can recover from overflow
GVL_System.RingBufferLog.ClearBuffer();
TestHandler.UpdateBufferHealthMetrics();

AssertEquals_REAL(
	Expected := 0.0,
	Actual := TestHandler.P_EventLogHandlerStatus.LoggingMetrics.BufferUtilizationPercentage,
	Delta := 0.01,
	Message := 'Buffer utilization should be 0% after clearing'
);

TEST_FINISHED();
END_METHOD

METHOD PRIVATE GivenPersistenceBlocked_WhenHandleFailureRuns_ExpectProcessingSuspendedUntilTimeout
VAR
END_VAR
TEST(__POUNAME());

//Assertions

TEST_FINISHED();
END_METHOD

METHOD PRIVATE GivenPersistenceThrowsException_WhenAddToEventLog_ExpectSafeRecovery
VAR
END_VAR
TEST(__POUNAME());

//Assertions

TEST_FINISHED();
END_METHOD

METHOD PRIVATE GivenProcessingAcrossAllSeverities_WhenMetricsUpdated_ExpectAccurateSeverityDistribution
VAR
END_VAR
TEST(__POUNAME());

//Assertions

TEST_FINISHED();
END_METHOD

METHOD PRIVATE GivenRestart_WhenLoggerResumes_ExpectMetricsResetAndSafeStartup
VAR
END_VAR
TEST(__POUNAME());

//Assertions

TEST_FINISHED();
END_METHOD

METHOD PRIVATE GivenBackoffTimerActive_WhenNextCycleRuns_ExpectNoPrematureRetries
VAR
END_VAR
TEST(__POUNAME());

//Assertions

TEST_FINISHED();
END_METHOD

METHOD PRIVATE GivenBufferAtMaxCapacity_WhenFloodedWithEntries_ExpectGracefulDegradation
VAR
END_VAR
TEST(__POUNAME());

//Assertions

TEST_FINISHED();
END_METHOD

METHOD PRIVATE GivenBufferOverflow_WhenRecovered_ExpectMetricsReflectCorrectDropCounts
VAR
END_VAR
TEST(__POUNAME());

//Assertions

TEST_FINISHED();
END_METHOD

METHOD PRIVATE GivenCycleExceeds_WhenDetected_ExpectHealthScoreReducedAndViolationLogged
VAR
END_VAR
TEST(__POUNAME());

//Assertions

TEST_FINISHED();
END_METHOD

METHOD PRIVATE GivenHeavyOSLoad_WhenPersistenceSlows_ExpectLoggerTaskStillMeetsCycleTime
VAR
END_VAR
TEST(__POUNAME());

//Assertions

TEST_FINISHED();
END_METHOD

METHOD PRIVATE GivenMaxDequeueRate_WhenCycleRuns_ExpectCycleTimeWithin50msBudget
VAR
END_VAR
TEST(__POUNAME());

//Assertions

TEST_FINISHED();
END_METHOD

METHOD PRIVATE GivenMixedSeverityFlood_WhenProcessing_ExpectLatencyForCriticalEntriesLow
VAR
END_VAR
TEST(__POUNAME());

//Assertions

TEST_FINISHED();
END_METHOD

METHOD PRIVATE GivenMultipleTasksMonitored_WhenSystemStable_ExpectUtilizationReportedAccurately
VAR
END_VAR
TEST(__POUNAME());

//Assertions

TEST_FINISHED();
END_METHOD

METHOD PRIVATE GivenPersistenceThrowsUnhandledException_WhenCaught_ExpectNoTaskCrash
VAR
END_VAR
TEST(__POUNAME());

//Assertions

TEST_FINISHED();
END_METHOD

METHOD PRIVATE GivenRepeatedPersistenceFailure_WhenRecovered_ExpectRateRestoredToNormal
VAR
END_VAR
TEST(__POUNAME());

//Assertions

TEST_FINISHED();
END_METHOD

METHOD PRIVATE GivenSeverityMix_WhenProcessing_ExpectSeverityDistributionAccurate
VAR
END_VAR
TEST(__POUNAME());

//Assertions

TEST_FINISHED();
END_METHOD

METHOD PRIVATE GivenSustainedHighThroughput_WhenRunningFor10Minutes_ExpectNoMemoryLeakOrCycleExceed
VAR
END_VAR
TEST(__POUNAME());

//Assertions

TEST_FINISHED();
END_METHOD

END_FUNCTION_BLOCK

// Tests/FB_RingBufferLoggerTests
FUNCTION_BLOCK FB_RingBufferLoggerTests EXTENDS TcUnit.FB_TestSuite
VAR
    i : DINT; //FOR loop index
    PointerBefore : PVOID;
    PointerAfter : PVOID;
    // Array instances for test methods (indices 0-57)
    RingBuffer : ARRAY[GC_Test.INDEX_TestFB_RingBuffer_MIN..GC_Test.INDEX_TestFB_RingBuffer_MAX] OF FB_RingBufferLogEntry;
END_VAR

GivenAdd3ObjectExpect3ObjectToBeAdded();
GivenAdd3Remove3ExpectFifoOrder();
GivenAddAndRemoveAlternateExpectFIFOOrder();
GivenAddExactCapacityThenRemoveAllExpectFIFO();
GivenAddMoreThanDoubleCapacityThenReadAllExpectOnlyRecent();
GivenRapidAddRemoveInLoopExpectCorrectFinalCount();
GivenAddObjectExpectStatusFlagsUpdateCorrectly();
GivenAddObjectLength10ExpectObjectToBeAdded();
GivenAddObjectLength20ExpectObjectToBeAdded();
GivenAddObjectLength40ExpectObjectToBeAdded();
GivenAddObjectLength80ExpectObjectToBeAdded();
GivenAddRemoveOneObjectExpectSameObjectBack();
GivenAddThenClearLastRemovedExpectEmptyFlag();
GivenAddThenQueryPointerConsistency();
GivenAddThenReadExpectSameObject();
GivenAddWhileRemoveInProgressExpectNoCorruption();
GivenAddWithinvalidRefExpectNoWrite();
GivenClearBufferExpectObjectCountZero();
GivenClearCalledExpectallStatsReset();
GivenEmptyBufferExpectPeekReturnsDefault();
GivenFullBufferAddOneExpectOverwriteOldest();
GivenLargeStringExpectTruncationOrError();
GivenMultipleAddinSingleCycleExpectAllStored();
GivenMultipleAddsSameCycleExpectAllStored();
GivenMultipleObjectsExpectPeekAlwaysReturnsFirst();
GivenNullRefInputExpectGracefulHandling();
GivenOneObjectAddedExpectPeekReturnsit();
GivenOversizedObjectExpectPartialWriteOrError();
GivenOverwriteOccursExpectOnlyRecentN();
GivenOverwriteThenReadExpectMostRecent();
GivenPeekThenClearPeekedFlagExpectReset();
GivenReadFromEmptyExpectNoCrashOrInvalid();
GivenReadThenClearStatusExpectFlagsReset();
GivenRemoveFromEmptyExpectError();
GivenRemoveObjectExpectLastRemovedMatchesExpected();
GivenRemoveOnEmptyExpectNoCrash();
GivenRemovePointerWrapsAroundExpectValidRead();
GivenRemoveThenReadExpectNoNewData();
GivenUpdateRemovePointerBoundaryExpectCorrectWrap();
GivenUpdateWritePointerBoundaryExpectCorrectWrap();
GivenWrapAroundReadPointerExpectCorrectRead();
GivenWrapAroundWriteExpectValidRead();
GivenWritePointerWrapsAroundExpectValidOverwrite();
GivenZeroCapacityBufferExpectNoWrite();
GivenInitExpectDefaultPointerAndState();
GivenAddThenRemoveExpectCorrectCounters();
GivenFillBufferExpectIsFullTrue();
GivenAddRemoveExpectFlagsSet();
GivenPeekAndReadExpectFlagsSet();
GivenOverwriteExpectFlagSet();
GivenAddExpectCorrectByteCount();
Test_BufferStatus_AfterAddAndRemove();
Test_BufferStatus_Add4Remove2();
GivenOverwriteThenRemoveExpectOverwriteCleared();
GivenAddMoreThanCapacityExpectCorrectGlobalCounter();
GivenReadThenRemoveExpectCorrectFlagsAndCounts();
GivenOversizedObject_WhenAdded_ExpectNoAdjacentMemoryCorruption();
GivenAddNullString_ExpectHandledGracefully();
GivenRemoveBeyondCapacity_ExpectSafeReset();
GivenOverwrite_WhenOccurs_ExpectDropCounterIncremented();
GivenWrapAroundManyTimes_ExpectCountersStable();

METHOD PRIVATE GivenAdd3ObjectExpect3ObjectToBeAdded
VAR
    TestObject      : ST_LogEntry := (Message := 'HelloWorld');
END_VAR
TEST(__POUNAME());

RingBuffer[0].Initialize();
RingBuffer[0].AddObject(RefObject := TestObject);
RingBuffer[0].AddObject(RefObject := TestObject);
RingBuffer[0].AddObject(RefObject := TestObject);

AssertEquals_UDINT(Actual := RingBuffer[0].RingBufferStatus.GlobalCounter, Expected := 3, 
            Message := 'Expected matching counts');

TEST_FINISHED();
END_METHOD

METHOD PRIVATE GivenAdd3Remove3ExpectFifoOrder
VAR
  Obj1 : ST_LogEntry := (Message := 'One');
  Obj2 : ST_LogEntry := (Message := 'Two');
  Obj3 : ST_LogEntry := (Message := 'Three');
  Removed : ST_LogEntry;
END_VAR
TEST(__POUNAME());

RingBuffer[1].Initialize();
RingBuffer[1].AddObject(RefObject := Obj1);
RingBuffer[1].AddObject(RefObject := Obj2);
RingBuffer[1].AddObject(RefObject := Obj3);

RingBuffer[1].RemoveObject(); Removed := RingBuffer[1].LastObjRemoved;
AssertEquals(Actual := Removed.Message, Expected := Obj1.Message, Message := 'First item should be "One"');

RingBuffer[1].RemoveObject(); Removed := RingBuffer[1].LastObjRemoved;
AssertEquals(Actual := Removed.Message, Expected := Obj2.Message, Message := 'Second item should be "Two"');

RingBuffer[1].RemoveObject(); Removed := RingBuffer[1].LastObjRemoved;
AssertEquals(Actual := Removed.Message, Expected := Obj3.Message, Message := 'Third item should be "Three"');

TEST_FINISHED();
END_METHOD

METHOD PRIVATE GivenAddAndRemoveAlternateExpectFIFOOrder
VAR
    TestObject : ST_LogEntry := (Message := 'Hello');
    Removed    : ST_LogEntry;
END_VAR
TEST(__POUNAME());

RingBuffer[2].Initialize();
RingBuffer[2].AddObject(RefObject := TestObject);
RingBuffer[2].RemoveObject(); Removed := RingBuffer[2].LastObjRemoved;
AssertEquals(Actual := Removed.Message, Expected := TestObject.Message,
    Message := 'Expected same object after alternate add/remove');
TEST_FINISHED();
END_METHOD

METHOD PRIVATE GivenAddExactCapacityThenRemoveAllExpectFIFO
VAR
    Capacity   : UDINT := RingBuffer[3].RingBufferStatus.BufferCapacity;
    i          : UDINT;
    Expected   : ST_LogEntry;
    Removed    : ST_LogEntry;
END_VAR
TEST(__POUNAME());

RingBuffer[3].Initialize();
Capacity := RingBuffer[3].RingBufferStatus.BufferCapacity;

// Add Capacity number of unique objects
FOR i := 1 TO Capacity DO
    Expected.Message := CONCAT('Item', UDINT_TO_STRING(i));
    RingBuffer[3].AddObject(RefObject := Expected);
END_FOR

// Remove and verify FIFO order
FOR i := 1 TO Capacity DO
    RingBuffer[3].RemoveObject();
    Removed := RingBuffer[3].LastObjRemoved;
    Expected.Message := CONCAT('Item', UDINT_TO_STRING(i));
    AssertEquals(Actual := Removed.Message, Expected := Expected.Message,
        Message := CONCAT('Expected FIFO order, mismatch at item ', UDINT_TO_STRING(i)));
END_FOR

TEST_FINISHED();
END_METHOD

METHOD PRIVATE GivenAddExpectCorrectByteCount
VAR
    TestObject  : ST_LogEntry := (Message := 'ByteCountTest');
    Expected    : ULINT;
END_VAR
TEST(__POUNAME());

RingBuffer[4].Initialize();
RingBuffer[4].AddObject(RefObject := TestObject);
Expected := RingBuffer[4].RingBufferConfiguration.ByteCountOfDataObj;

AssertEquals(
    Actual := RingBuffer[4].RingBufferStatus.ByteCountInBufferPrim,
    Expected := Expected,
    Message := 'Expected ByteCountInBufferPrim = ByteCountOfDataObj * 1'
);

TEST_FINISHED();
END_METHOD

METHOD PRIVATE GivenAddMaxUDINTObjectsExpectGracefulHandling
VAR
    TestObject : ST_LogEntry := (Message := 'Hello');
    Removed    : ST_LogEntry;
END_VAR
TEST(__POUNAME());

FOR i := 1 TO 100 DO
    RingBuffer[5].AddObject(RefObject := TestObject);
END_FOR

AssertTrue(Condition := RingBuffer[5].RingBufferStatus.GlobalCounter <= 100, Message := 'Buffer overflowed UDINT max unexpectedly');

TEST_FINISHED();
END_METHOD

METHOD PRIVATE GivenAddMoreThanCapacityExpectCorrectGlobalCounter
VAR
	DummyObj     : ST_LogEntry;
	i            : INT;
	capacity     : UDINT;
	testval80	: UDINT := 80;
END_VAR
TEST(__POUNAME());

RingBuffer[6].Initialize();
RingBuffer[6].ClearBuffer();
capacity := RingBuffer[6].RingBufferStatus.BufferCapacity;

// Add more than capacity to trigger overwriting
FOR i := 1 TO UDINT_TO_INT(capacity + 10) DO
	RingBuffer[6].AddObject(RefObject := DummyObj);
END_FOR

AssertEquals(capacity, RingBuffer[6].RingBufferStatus.GlobalCounter, 'Expected GlobalCounter to cap at capacity');
//AssertEquals(Expected := (testval80 * capacity), RingBuffer[6].RingBufferStat.ByteCountInBufferPrim, 'Expected ByteCount = capacity * size');
AssertTrue(RingBuffer[6].RingBufferStatus.Overwriting, 'Expected Overwriting = TRUE');

TEST_FINISHED();
END_METHOD

METHOD PRIVATE GivenAddMoreThanDoubleCapacityThenReadAllExpectOnlyRecent
VAR
    Capacity     : UDINT := RingBuffer[7].RingBufferStatus.BufferCapacity;
    TotalAdds    : UDINT := Capacity * 2 + 1;
    i            : UDINT;
    TestObject   : ST_LogEntry;
    Removed      : ST_LogEntry;
    ExpectedIdx  : UDINT;
    Expected     : ST_LogEntry;
END_VAR
TEST(__POUNAME());

// Add more than double the capacity worth of uniquely identifiable objects
FOR i := 1 TO TotalAdds DO
    TestObject.Message := CONCAT('Item', UDINT_TO_STRING(i));
    RingBuffer[7].AddObject(RefObject := TestObject);
END_FOR

// Only the most recent [Capacity] elements should be stored, starting from TotalAdds - Capacity + 1
FOR i := 1 TO Capacity DO
    RingBuffer[7].RemoveObject();
    Removed := RingBuffer[7].LastObjRemoved;
    ExpectedIdx := TotalAdds - Capacity + i;
    Expected.Message := CONCAT('Item', UDINT_TO_STRING(ExpectedIdx));
    AssertEquals(Actual := Removed.Message, Expected := Expected.Message,
        Message := CONCAT('Expected retained item: ', Expected.Message));
END_FOR

TEST_FINISHED();
END_METHOD

METHOD PRIVATE GivenAddNullString_ExpectHandledGracefully
VAR
    NullObject      : ST_LogEntry;
    ValidObject     : ST_LogEntry := (Message := 'ValidString');
    InitialCount    : UDINT;
    EmptyString     : STRING := '';
END_VAR
TEST(__POUNAME());

RingBuffer[58].Initialize();
RingBuffer[58].ClearBuffer();

// Get initial count
InitialCount := RingBuffer[58].RingBufferStatus.GlobalCounter;

// Test 1: Add object with null/empty string
NullObject.Message := EmptyString;
RingBuffer[58].AddObject(RefObject := NullObject);

// Should still add the object (empty string is valid)
AssertEquals_UDINT(
    Actual := RingBuffer[58].RingBufferStatus.GlobalCounter,
    Expected := InitialCount + 1,
    Message := 'Empty string object should be added'
);

// Test 2: Verify we can retrieve it
RingBuffer[58].RemoveObject();
AssertEquals(
    Actual := RingBuffer[58].LastObjRemoved.Message,
    Expected := EmptyString,
    Message := 'Should retrieve empty string correctly'
);

// Test 3: Mix null and valid strings
RingBuffer[58].AddObject(RefObject := NullObject);
RingBuffer[58].AddObject(RefObject := ValidObject);
RingBuffer[58].AddObject(RefObject := NullObject);

AssertEquals_UDINT(
    Actual := RingBuffer[58].RingBufferStatus.GlobalCounter,
    Expected := 3,
    Message := 'Should handle mix of empty and valid strings'
);

// Test 4: Verify FIFO order preserved
RingBuffer[58].RemoveObject();
AssertEquals(Actual := RingBuffer[58].LastObjRemoved.Message, Expected := EmptyString, Message := 'First empty string');

RingBuffer[58].RemoveObject();
AssertEquals(Actual := RingBuffer[58].LastObjRemoved.Message, Expected := ValidObject.Message, Message := 'Valid string');

RingBuffer[58].RemoveObject();
AssertEquals(Actual := RingBuffer[58].LastObjRemoved.Message, Expected := EmptyString, Message := 'Second empty string');

TEST_FINISHED();
END_METHOD

METHOD PRIVATE GivenAddObjectExpectStatusFlagsUpdateCorrectly
VAR
    TestObject : ST_LogEntry := (Message := 'StatusCheck');
END_VAR
TEST(__POUNAME());

RingBuffer[8].Initialize();

// Clear all status flags first
//fix
//RingBuffer[8].RingBufferStat.ObjectWasAddedPrimary := FALSE;
//RingBuffer[8].RingBufferStat.ObjectWasRemovedPrimary := FALSE;
//RingBuffer[8].RingBufferStat.ObjectWasPeekedPrimary := FALSE;

// Add an object
RingBuffer[8].AddObject(RefObject := TestObject);

// Assert that ObjectAddedPrimary is now TRUE
AssertTrue(
    Condition := RingBuffer[8].RingBufferStatus.ObjectWasAddedPrimary,
    Message := 'Expected ObjectAddedPrimary flag to be TRUE after AddObject()'
);

// Assert that other flags remain unaffected
AssertFalse(
    Condition := RingBuffer[8].RingBufferStatus.ObjectWasRemovedPrimary,
    Message := 'Expected ObjectRemovedPrimary flag to remain FALSE'
);

AssertFalse(
    Condition := RingBuffer[8].RingBufferStatus.ObjectWasPeekedPrimary,
    Message := 'Expected ObjectPeekedPrimary flag to remain FALSE'
);

TEST_FINISHED();
END_METHOD

METHOD PRIVATE GivenAddObjectLength10ExpectObjectToBeAdded
VAR
    TestObject      : ST_LogEntry := (Message := 'HelloWorld');  
END_VAR
TEST(__POUNAME());

RingBuffer[9].Initialize();
RingBuffer[9].AddObject(RefObject := TestObject);
RingBuffer[9].RemoveObject();

AssertEquals(Actual := RingBuffer[9].LastObjRemoved.Message, Expected := TestObject.Message,
            Message := 'Expected matching strings');

TEST_FINISHED();
END_METHOD

METHOD PRIVATE GivenAddObjectLength20ExpectObjectToBeAdded
VAR
    TestObject      : ST_LogEntry := (Message := 'HelloWorldHelloWorld');    
END_VAR
TEST(__POUNAME());

RingBuffer[10].Initialize();
RingBuffer[10].AddObject(RefObject := TestObject);
RingBuffer[10].RemoveObject();

AssertEquals(Actual := RingBuffer[10].LastObjRemoved.Message, Expected := TestObject.Message,
            Message := 'Expected matching strings');

TEST_FINISHED();
END_METHOD

METHOD PRIVATE GivenAddObjectLength40ExpectObjectToBeAdded
VAR
    TestObject      : ST_LogEntry := (Message := 'HelloWorldHelloWorldHelloWorldHelloWorld');    
END_VAR
TEST(__POUNAME());

RingBuffer[11].Initialize();
RingBuffer[11].AddObject(RefObject := TestObject);
RingBuffer[11].RemoveObject();

AssertEquals(Actual := RingBuffer[11].LastObjRemoved.Message, Expected := TestObject.Message,
            Message := 'Expected matching strings');

TEST_FINISHED();
END_METHOD

METHOD PRIVATE GivenAddObjectLength80ExpectObjectToBeAdded
VAR
    TestObject      : ST_LogEntry := (Message := 'HelloWorldHelloWorldHelloWorldHelloWorldHelloWorldHelloWorldHelloWorldHelloWorld');    
END_VAR
TEST(__POUNAME());

RingBuffer[12].Initialize();
RingBuffer[12].AddObject(RefObject := TestObject);
RingBuffer[12].RemoveObject();

AssertEquals(Actual := RingBuffer[12].LastObjRemoved.Message, Expected := TestObject.Message,
            Message := 'Expected matching strings');

TEST_FINISHED();
END_METHOD

METHOD PRIVATE GivenAddRemoveExpectFlagsSet
VAR
    TestObject  : ST_LogEntry := (Message := 'FlagTest');
END_VAR
TEST(__POUNAME());

RingBuffer[13].Initialize();
RingBuffer[13].AddObject(RefObject := TestObject);
AssertTrue(Condition := RingBuffer[13].RingBufferStatus.ObjectWasAddedPrimary, Message := 'Expected ObjectWasAddedPrimary = TRUE');

RingBuffer[13].RemoveObject();
AssertTrue(Condition := RingBuffer[13].RingBufferStatus.ObjectWasRemovedPrimary, Message := 'Expected ObjectWasRemovedPrimary = TRUE');

TEST_FINISHED();
END_METHOD

METHOD PRIVATE GivenAddRemoveOneObjectExpectSameObjectBack
VAR
  TestObject : ST_LogEntry := (Message := 'First');
  Removed : ST_LogEntry;
END_VAR
TEST(__POUNAME());

RingBuffer[14].Initialize();
RingBuffer[14].AddObject(RefObject := TestObject);
RingBuffer[14].RemoveObject();

Removed := RingBuffer[14].LastObjRemoved;

AssertEquals(Actual := Removed.Message, Expected := TestObject.Message, Message := 'Expected matching strings');

TEST_FINISHED();
END_METHOD

METHOD PRIVATE GivenAddThenClearLastRemovedExpectEmptyFlag
VAR

    TestObject : ST_LogEntry := (Message := 'ToBeRemoved');
	tempStr		: STRING := '';
END_VAR
TEST(__POUNAME());

RingBuffer[15].Initialize();
// Add and remove object to populate LastObjRemoved
RingBuffer[15].AddObject(RefObject := TestObject);
RingBuffer[15].RemoveObject();

// Verify LastObjRemoved is not empty
AssertEquals(
    Actual := RingBuffer[15].LastObjRemoved.Message,
    Expected := TestObject.Message,
    Message := 'Expected LastObjRemoved to contain the recently removed object'
);

// Clear LastObjRemoved
RingBuffer[15].ClearLastRemoved();

// Verify it has been cleared
AssertEquals(
    Actual := RingBuffer[15].LastObjRemoved.Message,
    Expected := tempStr,
    Message := 'Expected LastObjRemoved to be cleared (empty string)'
);

TEST_FINISHED();
END_METHOD

METHOD PRIVATE GivenAddThenQueryPointerConsistency
VAR

    TestObject : ST_LogEntry := (Message := 'Hello');
    WriteIndexBefore : UDINT;
    WriteIndexAfter  : UDINT;
END_VAR
TEST(__POUNAME());

RingBuffer[16].Initialize();

WriteIndexBefore := RingBuffer[16].WriteIndex;

RingBuffer[16].AddObject(RefObject := TestObject);

WriteIndexAfter := RingBuffer[16].WriteIndex;

AssertTrue(Condition := WriteIndexAfter <> WriteIndexBefore,
    Message := 'Expected write index to advance');

TEST_FINISHED();
END_METHOD

METHOD PRIVATE GivenAddThenReadExpectSameObject
VAR

    TestObject : ST_LogEntry;
    ReadObj    : ST_LogEntry;
    Obj1       : ST_LogEntry;
    Obj2       : ST_LogEntry;
    Obj3       : ST_LogEntry;
    Obj4       : ST_LogEntry;
END_VAR
TEST(__POUNAME());

RingBuffer[17].Initialize();
TestObject.Message := 'Alpha';
RingBuffer[17].AddObject(RefObject := TestObject);
RingBuffer[17].ReadObject();
ReadObj := RingBuffer[17].LastObjRead;
AssertEquals(Actual := ReadObj.Message, Expected := TestObject.Message,
             Message := 'Expected read value to match written value');
			 
TEST_FINISHED();
END_METHOD

METHOD PRIVATE GivenAddThenRemoveExpectCorrectCounters
VAR
    TestObject  : ST_LogEntry := (Message := 'CounterTest');
	testVal0	: UDINT :=0;
	testVal1	: UDINT :=1;
END_VAR
TEST(__POUNAME());

RingBuffer[18].Initialize();
RingBuffer[18].AddObject(RefObject := TestObject);
AssertEquals(Actual := RingBuffer[18].RingBufferStatus.GlobalCounter, Expected := testVal1, Message := 'Expected GlobalCounter = 1');
AssertEquals(Actual := RingBuffer[18].RingBufferStatus.ObjectCountInBufferPrim, Expected := testVal1, Message := 'Expected ObjectCount = 1');

RingBuffer[18].RemoveObject();
AssertEquals(Actual := RingBuffer[18].RingBufferStatus.GlobalCounter, Expected := testVal0, Message := 'Expected GlobalCounter = 0');
AssertEquals(Actual := RingBuffer[18].RingBufferStatus.ObjectCountInBufferPrim, Expected := testVal0, Message := 'Expected ObjectCount = 0');

TEST_FINISHED();
END_METHOD

METHOD PRIVATE GivenAddWhileRemoveInProgressExpectNoCorruption
VAR

    Obj1, Obj2, Obj3 : ST_LogEntry;
    Removed : ST_LogEntry;
END_VAR
TEST(__POUNAME());

RingBuffer[19].Initialize();
Obj1.Message := 'First';
Obj2.Message := 'Second';
Obj3.Message := 'Third';

// Add two objects
RingBuffer[19].AddObject(RefObject := Obj1);
RingBuffer[19].AddObject(RefObject := Obj2);

// Start a remove operation
RingBuffer[19].RemoveObject(); // Should remove Obj1

// Immediately add another object while remove has just happened
RingBuffer[19].AddObject(RefObject := Obj3);

// Remove again
RingBuffer[19].RemoveObject(); // Should remove Obj2
Removed := RingBuffer[19].LastObjRemoved;
AssertEquals(
    Actual := Removed.Message,
    Expected := Obj2.Message,
    Message := 'Expected second object to be removed correctly without corruption'
);

// Remove final object
RingBuffer[19].RemoveObject(); // Should remove Obj3
Removed := RingBuffer[19].LastObjRemoved;
AssertEquals(
    Actual := Removed.Message,
    Expected := Obj3.Message,
    Message := 'Expected third object to be removed correctly without corruption'
);

TEST_FINISHED();
END_METHOD

METHOD PRIVATE GivenAddWithInvalidRefExpectNoWrite
VAR

    TestObject : ST_LogEntry := (Message := 'Hello');
    Removed    : ST_LogEntry;
END_VAR
TEST(__POUNAME());

RingBuffer[20].Initialize();
TestObject.Message := 'ValidString';
RingBuffer[20].AddObject(RefObject := TestObject);

AssertEquals_UDINT(Actual := RingBuffer[20].RingBufferStatus.GlobalCounter, Expected := 1,
    Message := 'Expected valid string to be added');
	
TEST_FINISHED();
END_METHOD

METHOD PRIVATE GivenClearBufferExpectObjectCountZero
VAR

    TestObject : ST_LogEntry := (Message := 'Hello');
    Removed    : ST_LogEntry;
    testvalue   : UDINT := 0;
END_VAR
TEST(__POUNAME());

RingBuffer[21].AddObject(RefObject := TestObject);
RingBuffer[21].ClearBuffer();

AssertEquals(Actual := RingBuffer[21].RingBufferStatus.GlobalCounter, Expected := testvalue,
    Message := 'Expected cleared buffer to have zero object count');
	
TEST_FINISHED();
END_METHOD

METHOD PRIVATE GivenClearCalledExpectAllStatsReset
VAR

    Obj1, Obj2 : ST_LogEntry;
END_VAR
TEST(__POUNAME());

RingBuffer[22].Initialize();
Obj1.Message := 'Alpha';
Obj2.Message := 'Beta';

// Add two objects
RingBuffer[22].AddObject(RefObject := Obj1);
RingBuffer[22].AddObject(RefObject := Obj2);

// Remove one object to alter internal state
RingBuffer[22].RemoveObject();

// Now clear the buffer
RingBuffer[22].ClearBuffer();
RingBuffer[22].ClearStatusFlags();

// Check key stats are reset
AssertEquals_UDINT(
    Actual := RingBuffer[22].RingBufferStatus.GlobalCounter,
    Expected := 0,
    Message := 'Expected GlobalCounter to be reset to 0'
);

AssertEquals_LWORD(
    Actual := RingBuffer[22].pWrite,
    Expected := ADR(RingBuffer[22].Buffer[GPL_RingBuffer.MIN_LOGENTRIES]),
    Message := 'Expected write pointer to be reset to 0'
);

AssertEquals_LWORD(
    Actual := RingBuffer[22].pRemove,
    Expected := ADR(RingBuffer[22].Buffer[GPL_RingBuffer.MIN_LOGENTRIES]),
    Message := 'Expected remove pointer to be reset to 0'
);

AssertFalse(
    Condition := RingBuffer[22].RingBufferStatus.ObjectWasAddedPrimary,
    Message := 'Expected ObjectAddedPrimary to be cleared'
);

AssertFalse(
    Condition := RingBuffer[22].RingBufferStatus.ObjectWasRemovedPrimary,
    Message := 'Expected ObjectRemovedPrimary to be cleared'
);

AssertFalse(
    Condition := RingBuffer[22].RingBufferStatus.ObjectWasPeekedPrimary,
    Message := 'Expected ObjectPeekedPrimary to be cleared'
);

TEST_FINISHED();
END_METHOD

METHOD PRIVATE GivenCopyMemAreaValidInputExpectDataCopiedCorrectly
VAR

